(* CoDeSys 2.3.9.48 project: cy-wg-138-006.pro *)
(* Author: Avvitatrice doppia testa *)
(* Libraries: Standard.lib 20.5.14 07:13:26, Iecsfc.lib 16.5.13 13:00:50, SYSLIBCALLBACK.LIB 16.5.13 13:00:50, MBus_03.lib 9.2.13 16:51:58, mod_com.lib 16.5.13 13:00:50, Modb_l05.lib 13.5.15 09:30:08, SerComm.lib 16.5.13 13:00:50, Serial_Interface_01.lib 22.4.13 11:50:14, SysLibEvent.lib 16.5.13 13:00:50, SysLibFile.lib 16.5.13 13:00:50, SysLibPlcCtrl.lib 16.5.13 13:00:50, SysLibRtc.lib 16.5.13 13:00:50, SysLibSockets.lib 22.5.14 15:16:32, Util.lib 16.5.13 13:00:50, WagoLibMBX_01.lib 20.3.12 15:32:40, WagoLibModbus_IP_01.lib 24.7.13 14:05:58 *)

(* PLC configuration (modules and I/O channels)
0750-1506 8DI / 8DO 24V DC 0.5A [Type_34_8_Channels] node 1, in %IB144 out %QB144
  VPN_ST2 AT %IX72.0 [BOOLOnX_I] Ch_1 Digital input
  LAMP_AL AT %QX72.0 [BOOLOnX_Q] Ch_1 Digital output
  KEY_QE_ST AT %IX72.1 [BOOLOnX_I] Ch_2 Digital input
  AT %QX72.1 [BOOLOnX_Q] Ch_2 Digital output
  AT %IX72.2 [BOOLOnX_I] Ch_3 Digital input
  AT %QX72.2 [BOOLOnX_Q] Ch_3 Digital output
  AT %IX72.3 [BOOLOnX_I] Ch_4 Digital input
  AT %QX72.3 [BOOLOnX_Q] Ch_4 Digital output
  AT %IX72.4 [BOOLOnX_I] Ch_5 Digital input
  AT %QX72.4 [BOOLOnX_Q] Ch_5 Digital output
  AT %IX72.5 [BOOLOnX_I] Ch_6 Digital input
  AT %QX72.5 [BOOLOnX_Q] Ch_6 Digital output
  AT %IX72.6 [BOOLOnX_I] Ch_7 Digital input
  AT %QX72.6 [BOOLOnX_Q] Ch_7 Digital output
  AT %IX72.7 [BOOLOnX_I] Ch_8 Digital input
  AT %QX72.7 [BOOLOnX_Q] Ch_8 Digital output
0750-0652#48 RS-232/RS-485 Interface adjustable (48 Bytes) [Type_33_1_Channels] node 2, in %IB96 out %QB96
  AT %IB0 [BYTEOnB_I] First Byte of 48
  AT %QB0 [BYTEOnB_Q] First Byte of 48
0750-0652#48 RS-232/RS-485 Interface adjustable (48 Bytes) [Type_33_1_Channels] node 3, in %IB96 out %QB96
  AT %IB48 [BYTEOnB_I] First Byte of 48
  AT %QB48 [BYTEOnB_Q] First Byte of 48
0750-0652#48 RS-232/RS-485 Interface adjustable (48 Bytes) [Type_33_1_Channels] node 4, in %IB144 out %QB144
  AT %IB96 [BYTEOnB_I] First Byte of 48
  AT %QB96 [BYTEOnB_Q] First Byte of 48
Modbus variables [PFC200MODBUS] node 1, in %IB0 out %QB0 {PlcStopBehaviour = 1; FiledbusErrorBehaviour = 1; TcpOperation = 1; TcpPort = 502; TcpTimeout = 600; UdpOperation = 1; UdpPort = 502; RtuOperation = 0; NodeId = 1; ResponseTimeout = 5000; Interface = 0; Baud = 115200; StopBits = 1; Parity = 1; FlowCtrl = 0; PhysInterface = 0}
Modbus-Master [MB_MASTER] node 2, in %IB0 out %QB0
*)

(* Global variable list: Global_Constants *)
VAR_GLOBAL CONSTANT

	Plant_NAME			: STRING :='cySN:138 cyVER:138 - COIN Genova ';
	Plant_SN			: DWORD  :=138;	(* S/N Impianto di telecontrollo *)
	Plant_SW_VER		: WORD   :=1;		(* Versione SW installata *)


	(* Colour defines *)
	COLOR_RED			: DWORD	:= 16#2020F0;
	COLOR_YELLOW		: DWORD	:= 16#20F0F0;
	COLOR_GREEN			: DWORD	:= 16#20F020;
	COLOR_LIGHT_GREEN	: DWORD := 16#006000;

	(* Parameters *)
	Plant_DefaultTAmb	: INT	:=100;		(* [.1°C] Temperatura ambiente di default in caso di rottura sonda *)
	Plant_MaxRunTAmb	: INT   :=210; 		(* [.1°C] Temperatura ambiente massima funzionamento impianto *)
(*	Plant_AntiFreezeTAmb: INT   :=-40;		(* [.1°C] Antifreeze temperature, start circulators *)
	Plant_VRD_TAlarm	: INT   :=850; 		(* [.1°C] Temperatura di allarme VRD, blocco *)
	Plant_VRD_TMax		: INT   :=800; 		(* [.1°C] Setpoint massimo per uscita VRD *)
	Plant_VRD_TDefault	: INT	:=300;		(* [.1°C] Temperatura di default in caso di errore climatica *)
	Plant_CirOffDelay	: TIME	:=T#30m;	(* (Def.T#15m) Ritardo spegnimento pompe per ricircolo caldaia *)
	Plant_CirOnDelay	: TIME	:=T#15m;
	Plant_MaxWaterLoss	: WORD  :=2;		(* [lt/h] Massima perdita del circuito *) *)

	(* Filesystem *)
	FilesPath  			: STRING :='/media/sd/';(*'S:\'; *)

	(* TCP Logger *)
	Logger_SERVER		: STRING:='';
	Logger_IP			: STRING:='192.168.100.3';
	Logger_PORT			: WORD  :=80;
	Logger_GETSTART		: STRING:='GET /cygmsrv/hsgm.ashx?';
	Logger_GETEND		: STRING:='$R$N$R$N';
	Logger_CHECK		: STRING:='True';
	Logger_CRLF			: STRING:='$R$N';
	Logger_DataFile		: STRING:='/media/sd/LOG.DAT';
	Logger_DataFileOld	: STRING:='/media/sd/LOG.BCK';
	Logger_IndexFile	: STRING:='/media/sd/LOG.IDX';
	Logger_ConnRetries	: BYTE:=5;
	Logger_RecoverMsgs	: BYTE:=25;

	(* TCP Remote *)
	Remote_PORT			: WORD  :=10;
	Remote_WELCOME		: STRING:='Connected$R$N';
	Remote_OK			: STRING:='OK$R$N';
	Remote_ERROR		: STRING:='ERROR$R$N';

	(* TCP Sockets *)
	MAX_SEND_TCP_SERVER					 : DWORD:=60000;(*60000*)
	MAX_RECEIVE_TCP_SERVER				 : DWORD:=10000;
	MAX_RECEIVE_TCP_SERVER_SOCKET	 	 : DWORD:=2500;
	MAX_SEND_TCP_CLIENT					 : DWORD:=30000;(*15000*)
	MAX_RECEIVE_TCP_CLIENT				 : DWORD:=2500;
	MAX_RECEIVE_TCP_CLIENT_SOCKET		 : DWORD:=2500;
	MAX_RECEIVE_UDP_SERVER				 : INT  :=1472;
	MAX_RECEIVE_UDP_CLIENT				 : INT  :=1472;
	CONNECT_WATCHDOG_TIME				 : TIME :=t#10s;

END_VAR


VAR_GLOBAL
(*	TestNodoInterogato: BYTE;
	NodoDaInterrogare: BYTE;
	InibiscoModbus: BOOL;
 *)

	NodoDaInterrogareChiller: BYTE;
	InibiscoModbusChiller: BOOL;
	NodoDaInterrogareANZ: BYTE;
	InibiscoModbusANZ: BOOL;

	NodoDaInterrogareMB2: BYTE;
	InibiscoModbusMB2: BOOL;

	NodoDaInterrogareMB1: BYTE;
	InibiscoModbusMB1: BOOL;

	NodoDaInterrogareMB3: BYTE;
	InibiscoModbusMB3: BOOL;


END_VAR

VAR_GLOBAL RETAIN
	cmd_ControlMode_UTA01: BOOL;		(* variabili per abilitazione controllo UTA da CRONO o con comandi manuali da registro Modbus *)
	cmd_ControlMode_UTA02: BOOL;		(* variabili per abilitazione controllo UTA da CRONO o con comandi manuali da registro Modbus *)
	cmd_ControlMode_UTA03: BOOL;		(* variabili per abilitazione controllo UTA da CRONO o con comandi manuali da registro Modbus *)
	cmd_ControlMode_UTA04: BOOL;		(* variabili per abilitazione controllo UTA da CRONO o con comandi manuali da registro Modbus *)
	cmd_ControlMode_UTA05: BOOL;		(* variabili per abilitazione controllo UTA da CRONO o con comandi manuali da registro Modbus *)
	cmd_ControlMode_UTA06: BOOL;		(* variabili per abilitazione controllo UTA da CRONO o con comandi manuali da registro Modbus *)
	cmd_ControlMode_UTA07: BOOL;		(* variabili per abilitazione controllo UTA da CRONO o con comandi manuali da registro Modbus *)
	cmd_ControlMode_UTA08: BOOL;		(* variabili per abilitazione controllo UTA da CRONO o con comandi manuali da registro Modbus *)
	cmd_ControlMode_UTA09: BOOL;		(* variabili per abilitazione controllo UTA da CRONO o con comandi manuali da registro Modbus *)
	cmd_ControlMode_UTA10: BOOL;		(* variabili per abilitazione controllo UTA da CRONO o con comandi manuali da registro Modbus *)
	cmd_ControlMode_UTA12: BOOL;		(* variabili per abilitazione controllo UTA da CRONO o con comandi manuali da registro Modbus *)
	cmd_ControlMode_UTA13: BOOL;		(* variabili per abilitazione controllo UTA da CRONO o con comandi manuali da registro Modbus *)

END_VAR

(* Global variable list: Global_Retain *)
VAR_GLOBAL RETAIN PERSISTENT
(*	Mode_Manual : BOOL := FALSE; *)


(*	VRD01_Clima : typ_Clima;
	VRD02_Clima : typ_Clima;
	VRD03_Clima : typ_Clima;
	VRD04_Clima : typ_Clima; *)

	CHI01_Clima	: typ_Clima;
	CHI02_Clima	: typ_Clima;


(*	Ctl01_Counter	:	DWORD;
	Ctl02_Counter	:	DWORD; *)

(* Impostazioni di imipanto *)
(*
	DelayAllarmeTemperaturaNonRaggiunta: INT:=60;
	DeltaInterventoAllarmeTempeaturaNonRaggiuta: INT:=400;
	OffsetSetPointManuale:INT:=50;							(* Offset al Setpoint manuale per comensare lo scambiatore *)

	SogliaMinStartAntigelo: INT:=50;
	SogliaMinStopAntigelo: INT:=80;
	BitAbilitaAntigelo: BOOL:=TRUE;
*)

END_VAR

(* Global variable list: Global_Variables *)
VAR_GLOBAL

	SYS    : typ_SYS;
	Logger : typ_Logger;

	Lamp	:	LAMP_AL_GENERALE; (* Per gestione allarme generico impianto *)

	(**** PLANT OBJECTS ****)

	(* Frigo *)
	CHIAERMEC01	:obj_MODBUS_FRG_AER485P1 := (ID:=1, Address:=1);
	CHIAERMEC02	:obj_MODBUS_FRG_AER485P1 := (ID:=2, Address:=2);

	(* Cronothermostat *)
	THER01	:	obj_CRONTER_01 := (ID:=1, Local_MaxRunTAmb:=250,Histeresys:=10);
	THER02	:	obj_CRONTER_01 := (ID:=2, Local_MaxRunTAmb:=250,Histeresys:=10);
	THER03	:	obj_CRONTER_01 := (ID:=3, Local_MaxRunTAmb:=250,Histeresys:=10);
	THER04	:	obj_CRONTER_01 := (ID:=4, Local_MaxRunTAmb:=250,Histeresys:=10);
	THER05	:	obj_CRONTER_01 := (ID:=5, Local_MaxRunTAmb:=250,Histeresys:=10);
	THER06	:	obj_CRONTER_01 := (ID:=6, Local_MaxRunTAmb:=250,Histeresys:=10);
	THER07	:	obj_CRONTER_01 := (ID:=7, Local_MaxRunTAmb:=250,Histeresys:=10);
	THER08	:	obj_CRONTER_01 := (ID:=8, Local_MaxRunTAmb:=250,Histeresys:=10);
	THER09	:	obj_CRONTER_01 := (ID:=9, Local_MaxRunTAmb:=250,Histeresys:=10);
	THER10	:	obj_CRONTER_01 := (ID:=10, Local_MaxRunTAmb:=250,Histeresys:=10);
	THER12	:	obj_CRONTER_01 := (ID:=12, Local_MaxRunTAmb:=250,Histeresys:=10);
	THER13	:	obj_CRONTER_01 := (ID:=13, Local_MaxRunTAmb:=250,Histeresys:=10);


	CronEd	: 	obj_CRON_EDITOR_01;

	(* Gateway sonde Zeegbe *)

	GATEWAY	:	obj_GATEWAY_01 := (ID:=1, address:=1); 	(* gate way  *)


(* Sonde Tmperatura *)

	ZTHL01	:	obj_ZTHL_01 := (ID:=1, address:=16); 	(* Piano sotterraneo Rep. Bambino  *)
	ZTHL02	:	obj_ZTHL_01 := (ID:=2, address:=17); 	(* Piano sotterraneo Rep. Donna  *)
	ZTHL03	:	obj_ZTHL_01 := (ID:=3, address:=18); 	(* Piano terra ingresso - profumi   *)
	ZTHL04	:	obj_ZTHL_01 := (ID:=4, address:=19); 	(* Piano terra ingresso - rep. Uomo    *)
	ZTHL05	:	obj_ZTHL_01 := (ID:=5, address:=20);	(* Piano primo - reparto casa - lato cucina *)
	ZTHL06	:	obj_ZTHL_01 := (ID:=6, address:=21);	(* Piano primo - reparto casa - lato casse - uffici *)

(* Sonde CO2 *)

	COOV01	:	obj_COOV_01 := (ID:=1, address:=31); 	(* Piano sotterraneo Rep. Bambino  *)
	COOV02	:	obj_COOV_01 := (ID:=2, address:=32);	(* Piano sotterraneo Rep. Donna  *)
	COOV03	:	obj_COOV_01 := (ID:=3, address:=33);	(* Piano terra ingresso - profumi   *)
	COOV04	:	obj_COOV_01 := (ID:=4, address:=34);	(* Piano terra ingresso - rep. Uomo    *)
	COOV05	:	obj_COOV_01 := (ID:=5, address:=35);	(* Piano primo - reparto casa - lato cucina *)
	COOV06	:	obj_COOV_01 := (ID:=6, address:=36);	(* Piano primo - reparto casa - lato casse - uffici *)


	ANZ01	:	obj_MODBUS_FRER_QUBOH:= (ID:=1,Address:=1);	(* Generale  *)
	ANZ02	:	obj_MODBUS_FRER_QUBOH := (ID:=2,Address:=2);	(* QE. Uffici - QU  *)
	ANZ03	:	obj_MODBUS_FRER_QUBOH:= (ID:=3,Address:=3);	(* Gruppo frigo 1  *)
	ANZ04	:	obj_MODBUS_FRER_QUBOH:= (ID:=4,Address:=4);	(* Gruppo frigo 2  *)
	ANZ05	:	obj_MODBUS_FRER_QUBOH:= (ID:=5,Address:=5);	(* Q.E. UTA 1-5  *)
	ANZ06	:	obj_MODBUS_FRER_QUBOH:= (ID:=6,Address:=6);	(* Linee UTA (n.3 - una per fase) *)
	ANZ07	:	obj_MODBUS_FRER_QUBOH:= (ID:=7,Address:=7);	(* Linee UTA (n.3 - una per fase) *)
	ANZ08	:	obj_MODBUS_FRER_QUBOH:= (ID:=8,Address:=8);	(* Linee UTA (n.2 - una per fase) *)


	TREND : obj_MODBUS_TRENDCOIN_01 := (ID:=1,Address:=1);


(*** UTA ***)

	UTA01  	: obj_UTA_02:=(ID:=1);
	UTA02  	: obj_UTA_02:=(ID:=2);
	UTA03  	: obj_UTA_02:=(ID:=3);
	UTA04  	: obj_UTA_02:=(ID:=4);
	UTA05  	: obj_UTA_02:=(ID:=5);
	UTA06  	: obj_UTA_02:=(ID:=6);
	UTA07  	: obj_UTA_02:=(ID:=7);
	UTA08  	: obj_UTA_02:=(ID:=8);
	UTA09  	: obj_UTA_02:=(ID:=9);
	UTA10  	: obj_UTA_02:=(ID:=10);
(*	UTA11  	: obj_UTA_02:=(ID:=11); *)
	UTA12  	: obj_UTA_02:=(ID:=12);
	UTA13  	: obj_UTA_02:=(ID:=13);


	(** Communication **)
	(* ModBus *)

	MODB01	:	obj_MODBUS		:= (ID:=1, COM:=0, BAUDRATE:=BAUD_19200,RS485:=TRUE,MB_timeOut:=t#500ms);
	MODB02	:	obj_MODBUS		:= (ID:=2, COM:=2, BAUDRATE:=BAUD_9600 ,N_STOPBits:=2,RS485:=TRUE,MB_timeOut:=t#500ms);
	MODB03	:	obj_MODBUS 		:= (ID:=3, COM:=3, BAUDRATE:=BAUD_19200,N_STOPBits:=2,RS485:=TRUE,MB_timeOut:=t#500ms);
	MODB04	:	obj_MODBUS 		:= (ID:=4, COM:=4, BAUDRATE:=BAUD_19200,N_STOPBits:=2,RS485:=TRUE,MB_timeOut:=t#500ms);


	(**** SIMULATION ONLY ****)

	AggiornaLog: BOOL;

	(*...*)


END_VAR

(* Data type in Logger *)
TYPE en_Logger_ErrLev :
(
	EL_Log			:=0,
	EL_Wrn			:=1,
	EL_Alarm		:=2,
	EL_AlarmStop	:=3
);
END_TYPE

(* Data type in Logger *)
TYPE en_Logger_Status :
(
	S_Logger_UNKNOWN := 0,
	S_Logger_IDLE,
	S_Logger_WAITCONN,
	S_Logger_WAITTX,
	S_Logger_WAITRESP,
	S_Logger_ERROR
);
END_TYPE

(* Data type *)
TYPE en_SYS_Objects :
(
	EO_SYS		:=0,  (* PLC *)
	EO_VPN		:=1,  (* VPN *)
	EO_DOOR		:=2,  (* Door & access control *)

	EO_CAL		:=10, (* Caldaia *)
	EO_CIR		:=11, (* Circolatore *)
	EO_CRON		:=12, (* Crono-termostato *)
	EO_VRD		:=13, (* Valvola miscelatore pannelli *)
	EO_CTL		:=14, (* Contalitri *)
	EO_CTB		:=15, (* Contabilizzatore *)
	EO_TPV		:=16, (* Temperature probes values *)
	EO_PPV		:=17, (* Pressure probes values *)
	EO_PBV		:=18, (* Over-Pressure Alarms *)
	EO_TBV		:=19, (* Over-Temperature Alarms *)
	EO_PMV		:=20, (* Under-Pressure Alarms *)
	EO_GRU		:=21, (* Gruppo termico *)
	EO_PDC		:=22, (* Pompa di calore *)
	EO_SOL		:=23, (* Pannello solare termico *)
	EO_ESOL		:=24, (* Pannello solare fotovoltaico *)
	EO_GAS		:=25, (* Contatore GAS *)
	EO_PORT		:=26, (* Misuratore di portata *)
	EO_FPV		:=27, (* Flow probes values *)
	EO_ANZ		:=28, (* Analizzatore di rete *)
	EO_SCA		:=29, (* Signal Control Alarms *)
	EO_LUX		:=30, (* Base Illumination point *)
	EO_LUXM		:=31, (* Metered Illumination point *)
	EO_PSG		:=32, (* Sensore di passaggio *)
	EO_HVAC		:=33, (* Heating, Ventilating and Air Conditioning *)
	EO_HYGRV	:=34, (* Relative Humidity sensors value *)
	EO_COOV		:=35, (* Carbon Dioxide CO2 sensors value *)
	EO_INV		:=36, (* Inverter *)
	EO_STR		:=37, (* Smart string box *)

	EO_CIRD		:=39, (* Double CIR *)
	EO_ACS		:=40, (* Hot domestic water *)
	EO_CHI		:=41, (* Chiller *)
	EO_THER		:=42, (* Thermostat *)
	EO_CIRM		:=43, (* Modbus CIR *)
	EO_CIRDM	:=44, (* Modbus double CIR *)


	EO_UTA		:=47, (* UTA  *)
	EO_CHIAERMEC:=48, (* Frigorifero Aermec *)
	EO_UTACOIN	:=49, (* UTA  *)
	EO_POOL	:=50, 		(* Mischiotto  *)
	EO_ZCOOV:= 51, 		(*Sonda C02 Zigbee ZCOOVxxx *)


	EO_ZGW			:=200,  (* ZigBee - Gateway *)
	EO_ZRM			:=201,	(* ZigBee - Repeater *)
	EO_ZREL			:=202,	(* ZigBee - Actuator rele *)
	EO_ZTHL			:=203,	(* ZigBee - Temperature Sensor *)

	EO_ASGW			:=250,	(* ASi - Gateway *)
	EO_ASCBI		:=251,	(* ASi - Input Board, Ciabatta *)

	EO_LON			:=1000, (* Bus - LON *)
	EO_MODBUS		:=1001, (* Bus - MODBUS *)
	EO_MBUS			:=1002, (* Bus - M-BUS *)
	EO_MODBUS_TCP	:=1003, (* Bus - MODBUS TCP *)

	EO_GENERIC		:=9000, (* Generic dataset *)
	EO_EXPO			:=9001 (* EXPO dataset *)
);
END_TYPE

(* Data type *)
TYPE en_SYS_Status :
(
	S_UNKNOWN  := 0,
	S_STARTUP,
	S_INIT_RTC,
	S_INIT_VAR,
	S_AUTOTEST,
	S_RUNNING,
	S_SHUTDOWN,
	S_HALT
);
END_TYPE

(* Data type in Plant_Objects *)
TYPE typ_Clima : (* CURVA CLIMATICA *)
STRUCT
	InitOK:		BOOL;
	Points: 	ARRAY [0..10] OF POINT;
END_STRUCT
END_TYPE

(* Data type in Plant_Objects *)
TYPE typ_Cron_Calendar :
STRUCT
	Profile		: ARRAY[0..384] OF BYTE;
END_STRUCT
END_TYPE

(* Data type in Plant_Objects *)
TYPE typ_Cron_Jolly :
STRUCT
	Start		: DT;
	End			: DT;
	Temp		: WORD;
	Flags		: WORD; (* B0:Enabled B1..B15:Unused *)
END_STRUCT
END_TYPE

(* Data type in Plant_Objects *)
TYPE typ_Cron_Profile :
STRUCT
	Flags		: WORD;
	Setpoint	: ARRAY [0..95] OF WORD;
END_STRUCT
END_TYPE

(* Data type in Plant_Objects *)
TYPE typ_Frigo :
STRUCT
	Status	:	BOOL;		(* 0=OFF, 1=ON	*)
	Mode	:	BOOL;		(* 0=COLD, 1=HOT	*)
	Reset	:	BOOL;		(* 1=RESET	*)

	Alarm	:	DWORD;		(* 30 alarms of type bool grouped in one variable of 32 bits (last 2 don't used) *)

	(*  ALARM CODE (bit order of dword "Alarm": first is bit 0, last bit29)
        8	:	Allarme flussostato
		9	:	Allarme termica pompa condensante 
		10	:	Allarme termica pompa evaporante 
		11	:	Allarme resa 
		12	:	Allarme termica compressore circuito 1 
		13	:	Allarme bassa pressione circuito 1
		14	:	Allarme alta pressione circuito 1 
		15	:	Allarme antigelo circuito 1	
		16	:	Allarme termica ventilatore circuito 1	
		17	:	Allarme pressostato olio crcuito 1	
		18	:	Allarme sonda circuito 1	
		19	:	Allarme termica compressore circuito 2	
		20	:	Allarme bassa pressione circuito 2	
		21	:	Allarme alta pressione circuito 2	
		22	:	Allarme antigelo circuito 2	
		23	:	Allarme termica ventilatore circuito 2	
		24	:	Allarme pressostato olio circuito 2	
		25	:	Allarme sonda circuito 2	
		26	:	Allarme monitor tensione	
		27	:	Allarme pumpdown circuito 1	
		28	:	Allarme pumpdown circuito 2	
		29	:	Allarme eeprom	
		30	:	Allarme clock calendar	
		80	:	Allarme flussostato recuperatore	
		81	:	Allarme termica compressore circuito 1A	
		82	:	Allarme termica compressore circuito 1B	
		83	:	Allarme termica pompa evaporatore 1	
		84	:	Allarme termica pompa evaporatore 2	
		85	:	Allarme termica pompa evaporatore 3	
		86	:	Allarme antigelo evaporatore circuito 1	
		87	:	Allarme antigelo evaporatore circuito 2	
	*)


END_STRUCT
END_TYPE

(* Data type in Logger *)
TYPE typ_Logger :
STRUCT
	Status		: en_Logger_Status;

	SendReq		: BOOL;
	SendIdx		: DWORD;
	SendData	: ARRAY [0..MAX_SEND_TCP_CLIENT] OF BYTE;
	SendLen		: DINT;

	TData		: ARRAY [0..MAX_SEND_TCP_CLIENT] OF BYTE;
	TLen		: DINT;

	LastIdxPos	: DWORD;

	(* Temporary variables used by objects *)
	s1			: STRING(256);
	i1			: WORD;

END_STRUCT
END_TYPE

(* Data type in Plant_Objects *)
TYPE typ_MODBUS_CIR :
STRUCT
	PumpStatus		:	WORD;
	PumpFault		:	BOOL;
	PumpBoardTemp	:	INT;	(* Electonic board temperature  [°C] *)
	PumpVoltage		:	WORD;	(* Input voltage rms [V] *)
	PumpCurrent		:	WORD;	(* Output current [E-3 A]	*)
	PumpRPM			:	WORD;	(* Round per minute [rpm] *)
	PumpPower		:	WORD;	(* Power [W] *)
	PumpOpTime		:	DWORD;	(* Pump operating time [h] *)
	PumpHead		:	WORD;	(* [E-1 m] *)
	PumpFlow		:	WORD;	(* Extimated flow [E-1 m3/h] *)
	PumpLiqTemp		:	WORD;	(* Liquid temperature [°C] *)
	PumpAlarm		:	ARRAY [0..14] OF WORD;

END_STRUCT
END_TYPE

(* Data type in Plant_Objects *)
TYPE typ_MODBUS_FRER_QUBOH :
STRUCT
	V_L1N		:	DINT;	(* E-3 V *)
	V_L2N		:	DINT;
	V_L3N		:	DINT;
	V_L1L2		:	DINT;
	V_L2L3		:	DINT;
	V_L3L1		:	DINT;
	I_L1			:	DINT;	(* E-3 A *)
	I_L2			:	DINT;
	I_L3			:	DINT;

	FREQ		:	DWORD;	(* E-3 Hz *)

	P_3P			:	DINT;	(* W *)
	Q_3P		:	DINT;	(* VAr *)
	PF_3P		:	DINT;	(* E-3 *)
	WH_3P		:	DINT;	(* Wh *)
	VARH_3P		:	DINT;	(* VArh *)
	Multiplier	:	DWORD;

	V_3P		:	DINT;	(* E-3 V *)
	I_3P		:	DINT;	(* E-3 A *)

	COS_3P		:	DINT;	(* E-3 *)

	VA_3P		:	DINT;	(* VA *)
	P_L1		:	DWORD;	(* W *)
	P_L2		:	DWORD;
	P_L3		:	DWORD;
	Q_L1		:	DINT;	(* VAr *)
	Q_L2		:	DINT;
	Q_L3		:	DINT;
	VA_L1		:	DINT;	(* VA *)
	VA_L2		:	DINT;
	VA_L3		:	DINT;
	PF_L1		:	DINT;	(* E-3 *)
	PF_L2		:	DINT;
	PF_L3		:	DINT;
	COS_L1		:	DINT;	(* E-3 *)
	COS_L2		:	DINT;
	COS_L3		:	DINT;

	P_3P_Max	:	DINT;	(* W *)
	P_3P_Avg		:	DINT;

	I_L1_Max	:	DINT;	(* E-3 A *)
	I_L2_Max	:	DINT;
	I_L3_Max	:	DINT;

	Q_3P_Max	:	DINT;	(* VAr *)

END_STRUCT
END_TYPE

(* Data type in Plant_Objects *)
TYPE typ_MODBUS_VAR : (* Gestione parametri MODBUS *)
STRUCT
	SlaveAddress	: BYTE;
	FunCode			: BYTE;
	FunAddress		: WORD;
	Refresh_Time	: BYTE; (* 0:No refresh x:Refresh in seconds *)
	Refresh_Cnt		: BYTE; (* INTERNAL *)
	Variable		: POINTER TO WORD;
	Variable_Size	: BYTE;
	Variable_Mirror : WORD; (* INTERNAL [Force refresh on read variables when <>0] *)
END_STRUCT
END_TYPE

(* Data type *)
TYPE typ_SYS :
STRUCT
	Status			: en_SYS_Status;
	Warning			: BOOL;
	Alarm			: BOOL;
	AlarmStop		: BOOL;

	Time_LogString	: STRING;
	Time_Year		: WORD;
	Time_Month		: BYTE;
	Time_Day		: BYTE;
	Time_Hour		: BYTE;
	Time_Minute		: BYTE;

	Time_CT_DT		: DT;
	Time_CT_Day		: WORD;
	Time_CT_Quarter	: BYTE;

	LastLogs_Idx	: BYTE;
	LastLogs_Dat	: ARRAY[0..5] OF STRING;
	LastLogs_Msg	: ARRAY[0..5] OF STRING;

END_STRUCT
END_TYPE

(* Data type in Plant_Objects *)
TYPE typ_VisuStrutturaMbus :
STRUCT

	sdNodoPresente: STRING(16);
	sdEnergia: STRING(16);
	sdPotenza: STRING(16);
	sdVolume: STRING(16);
	sdFlow: STRING(16);
	sdTempIngresso: STRING(8);
	sdTempaUscita: STRING(8);
	sdTempDelta: STRING(8);

END_STRUCT
END_TYPE

(* POU PLC_PRG, ST *)
PROGRAM PLC_PRG
VAR
	Timer1: TON; (* Fast controls tick *)
	Timer2: TON; (* Plant control tick *)
	Timer3: TON; (* Logger timer *)

	i : INT;

	R_TRIG_CHIAERMEC01_ScriviDato: F_TRIG;
	R_TRIG_CHIAERMEC02_ScriviDato: F_TRIG;
	R_TRIG_TREND_ScriviDato: F_TRIG;

	aggiornalogdaModBus: BOOL;
	tonaggiornaLogdaModBus: TON;
	EseguiLog: INT;
	Ton_pausaTrig: TON;
	s1: STRING;
	R_TrigAggiornaLog: R_TRIG;
	allarme,warning:BOOL;
END_VAR
VAR_INPUT
	RichiestaLogDaRemoto: BOOL;
END_VAR
(******************************************************************************
 ****                           MAIN TASK CODE                             ****
 ******************************************************************************

	Network setup:
		IP  = 192.168.100.2 | MSK = 255.255.255.0
		GW	= 192.168.100.1 | DNS = 192.168.100.1
		SNTP = 193.204.114.232 (3600s) ==> 192.168.100.3

*)

(*==============================*)
(*===== Main status machine ====*)
(*==============================*)
Main_Stm();

(*==============================*)
(*== Running cycle operations ==*)
(*==============================*)
IF SYS.Status>S_INIT_VAR THEN
	(* Execute cycle processes *)


	MODB01();
(*	TREND(ModBus:=MODB01,
			ScriviRUN_UTA01:=UTA01.cmd_DO_OUT,
			ScriviRUN_UTA02:=UTA02.cmd_DO_OUT,
			ScriviRUN_UTA03:=UTA03.cmd_DO_OUT,
			ScriviRUN_UTA04:=UTA04.cmd_DO_OUT,
			ScriviRUN_UTA05:=UTA05.cmd_DO_OUT,
			ScriviRUN_UTA06:=UTA06.cmd_DO_OUT,
			ScriviRUN_UTA07:=UTA07.cmd_DO_OUT,
			ScriviRUN_UTA08:=UTA08.cmd_DO_OUT,
			ScriviRUN_UTA09:=UTA09.cmd_DO_OUT,
			ScriviRUN_UTA10:=UTA10.cmd_DO_OUT,
			ScriviRUN_UTA12:=UTA12.cmd_DO_OUT,
			ScriviRUN_UTA13:=UTA13.cmd_DO_OUT,
			); *)




	TREND(ModBus:=MODB01);

	TREND(
			ControlMode_UTA01:=cmd_ControlMode_UTA01,
 			ControlMode_UTA02:=cmd_ControlMode_UTA02,
			ControlMode_UTA03:=cmd_ControlMode_UTA03,
			ControlMode_UTA04:=cmd_ControlMode_UTA04,
			ControlMode_UTA05:=cmd_ControlMode_UTA05,
			ControlMode_UTA06:=cmd_ControlMode_UTA06,
			ControlMode_UTA07:=cmd_ControlMode_UTA07,
			ControlMode_UTA08:=cmd_ControlMode_UTA08,
			ControlMode_UTA09:=cmd_ControlMode_UTA09,
			ControlMode_UTA10:=cmd_ControlMode_UTA10,
			ControlMode_UTA12:=cmd_ControlMode_UTA12,
			ControlMode_UTA13:=cmd_ControlMode_UTA13,
			ScriviRUN_UTA01:=UTA01.cmd_DO_OUT ,
			ScriviRUN_UTA02:=UTA02.cmd_DO_OUT ,
			ScriviRUN_UTA03:=UTA03.cmd_DO_OUT ,
			ScriviRUN_UTA04:=UTA04.cmd_DO_OUT ,
			ScriviRUN_UTA05:=UTA05.cmd_DO_OUT ,
			ScriviRUN_UTA06:=UTA06.cmd_DO_OUT ,
			ScriviRUN_UTA07:=UTA07.cmd_DO_OUT ,
			ScriviRUN_UTA08:=UTA08.cmd_DO_OUT ,
			ScriviRUN_UTA09:=UTA09.cmd_DO_OUT ,
			ScriviRUN_UTA10:=UTA10.cmd_DO_OUT ,
			ScriviRUN_UTA12:=UTA12.cmd_DO_OUT ,
			ScriviRUN_UTA13:=UTA13.cmd_DO_OUT ,
			ScriviSP_UTA01:=UTA01.cmd_DO_SetPoint ,
			ScriviSP_UTA02:=UTA02.cmd_DO_SetPoint ,
			ScriviSP_UTA03:=UTA03.cmd_DO_SetPoint ,
			ScriviSP_UTA04:=UTA04.cmd_DO_SetPoint ,
			ScriviSP_UTA05:=UTA05.cmd_DO_SetPoint ,
			ScriviSP_UTA06:=UTA06.cmd_DO_SetPoint ,
			ScriviSP_UTA07:=UTA07.cmd_DO_SetPoint ,
			ScriviSP_UTA08:=UTA08.cmd_DO_SetPoint ,
			ScriviSP_UTA09:=UTA09.cmd_DO_SetPoint ,
			ScriviSP_UTA10:=UTA10.cmd_DO_SetPoint ,
			ScriviSP_UTA12:=UTA12.cmd_DO_SetPoint ,
			ScriviSP_UTA13:=UTA13.cmd_DO_SetPoint ,
			ModBus:=MODB01 ,
			Status_Log=> ,
			Status_Vis=> );


	NodoDaInterrogareMB1:=1;

UTA01(
	UTA_ST:=TREND.MB_BitStatoCoil[19],
	UTA_CentrAL:=TREND.MB_BitStato[102] OR TREND.MB_BitStato[103],   (* TRUE= Flusso , FALSE = No Flusso *)
	T_AMB:=TREND.MB_RegistriLetti[134] ,
	UR_AMB:=TREND.MB_RegistriLetti[135]  ,
	T_MISC:=TREND.MB_RegistriLetti[136]  ,
	UR_MISC:=TREND.MB_RegistriLetti[137]  ,
	T_MAND:=TREND.MB_RegistriLetti[138]  ,
	T_EST:=TREND.MB_RegistriLetti[139]  ,
	UR_EST:= TREND.MB_RegistriLetti[140] ,
	ENTALPIA_EST:=TREND.MB_RegistriLetti[141]  ,
	ENTALPIA_AMB:=TREND.MB_RegistriLetti[142] ,
	UMID_ASS_EST:=TREND.MB_RegistriLetti[143]  ,
	UMID_ASS_AMB:= TREND.MB_RegistriLetti[144] ,
	UMID_ASS_MISC:=TREND.MB_RegistriLetti[145] ,
	UMID_ASS_CONDEN:=TREND.MB_RegistriLetti[146]  ,
	SET_COMP_T_AMB:=TREND.MB_RegistriLetti[147]  ,
	RITAR_SET_T_AMB:= TREND.MB_RegistriHoldingLetti[68],
	SET_T_MAND:= TREND.MB_RegistriHoldingLetti[69] ,
	SET_ANTIGELO:= TREND.MB_RegistriHoldingLetti[70] ,
	SET_UR_AMB:= TREND.MB_RegistriHoldingLetti[71],
	ISTERESI_UR_AMB:= TREND.MB_RegistriHoldingLetti[72] ,
	SET_F_ANTIG_AMB:= TREND.MB_RegistriHoldingLetti[73] ,
	SOGLIA_T_EST_VR:=  TREND.MB_RegistriHoldingLetti[74],
	MIN_AP_SERR_E_R:=  TREND.MB_RegistriHoldingLetti[75],
	MIN_AP_SERR_ESP:=  TREND.MB_RegistriHoldingLetti[76],
	RID_SET_T_RISC:=  TREND.MB_RegistriHoldingLetti[77],
	VENT_MAND:= TREND.MB_BitStato[141],
	VENT_RIPR:=TREND.MB_BitStato[142] ,
	P_UMIDIF:=TREND.MB_BitStato[143] ,
	VALV_B_FREDDA:=TREND.MB_BitStato[151] ,
	VALV_B_CALDA:=TREND.MB_BitStato[152] ,
	SERRANDE_ESP:= TREND.MB_BitStato[153],
	SERRAND_EST_RIC:= TREND.MB_BitStato[154],
	ABILITA:=TREND.MB_BitStatoCoil[19] ,
	STATO_VENT_M:=TREND.MB_BitStato[99] ,
	STATO_VENT_R:=TREND.MB_BitStato[100] ,
	FILTRO:=TREND.MB_BitStato[101] ,
	FLUSSO_VM:=TREND.MB_BitStato[102] ,
	FLUSSO_VR:= TREND.MB_BitStato[103],
	FILTRI_INTASATI:= TREND.MB_BitStato[104],
	ALL_VERIFICA_VM:=TREND.MB_BitStato[105] ,
	ALL_VERIFICA_VR:= TREND.MB_BitStato[106],
	ALL_V011_MANC_SPEGN:= TREND.MB_BitStato[107],
	ALL_V011_MANC_FUNZ:=TREND.MB_BitStato[108],
	ALL_V012_MANC_SPEGN:=TREND.MB_BitStato[109] ,
	ALL_V012_MANC_FUNZ:=TREND.MB_BitStato[110],
	cmd_DI_RUN:=THER01.RunCrono,
	cmd_DI_SetPoint:=THER01.SetPoint,
	UTA_CONTROL_MODE:=cmd_ControlMode_UTA01	);



	UTA02(
	UTA_ST:= TREND.MB_BitStatoCoil[20],     	(* ABILITA UTA  *)
	UTA_CentrAL:=TREND.MB_BitStato[120] OR TREND.MB_BitStato[121],	 (* TRUE= Flusso , FALSE = No Flusso *)
	T_AMB:=TREND.MB_RegistriLetti[155] ,
	UR_AMB:=TREND.MB_RegistriLetti[156]  ,
	T_MISC:=TREND.MB_RegistriLetti[157]  ,
	UR_MISC:=TREND.MB_RegistriLetti[158]  ,
	T_MAND:=TREND.MB_RegistriLetti[159]  ,
	T_EST:=TREND.MB_RegistriLetti[165]  ,
	UR_EST:= TREND.MB_RegistriLetti[166] ,
	ENTALPIA_EST:=TREND.MB_RegistriLetti[169]  ,
	ENTALPIA_AMB:=TREND.MB_RegistriLetti[170] ,
	UMID_ASS_EST:=TREND.MB_RegistriLetti[171]  ,
	UMID_ASS_AMB:= TREND.MB_RegistriLetti[172] ,
	UMID_ASS_MISC:=TREND.MB_RegistriLetti[173] ,
	UMID_ASS_CONDEN:=TREND.MB_RegistriLetti[174]  ,
	SET_COMP_T_AMB:=TREND.MB_RegistriLetti[167]  ,
	RITAR_SET_T_AMB:= TREND.MB_RegistriHoldingLetti[78],
	SET_T_MAND:= TREND.MB_RegistriHoldingLetti[79] ,
	SET_ANTIGELO:= TREND.MB_RegistriHoldingLetti[80] ,
	SET_UR_AMB:= TREND.MB_RegistriHoldingLetti[81],
	ISTERESI_UR_AMB:= TREND.MB_RegistriHoldingLetti[82] ,
	SET_F_ANTIG_AMB:= TREND.MB_RegistriHoldingLetti[83] ,
	SOGLIA_T_EST_VR:=  TREND.MB_RegistriHoldingLetti[84],
	MIN_AP_SERR_E_R:=  TREND.MB_RegistriHoldingLetti[85],
	MIN_AP_SERR_ESP:=  TREND.MB_RegistriHoldingLetti[86],
	RID_SET_T_RISC:=  TREND.MB_RegistriHoldingLetti[87],
	VENT_MAND:= TREND.MB_BitStato[111],
	VENT_RIPR:=TREND.MB_BitStato[112] ,
	P_UMIDIF:=TREND.MB_BitStato[113] ,
	VALV_B_FREDDA:=TREND.MB_BitStato[181] ,
	VALV_B_CALDA:=TREND.MB_BitStato[182] ,
	SERRANDE_ESP:= TREND.MB_BitStato[183],
	SERRAND_EST_RIC:= TREND.MB_BitStato[184],
	ABILITA:=TREND.MB_BitStatoCoil[20] ,
	STATO_VENT_M:=TREND.MB_BitStato[117] ,
	STATO_VENT_R:=TREND.MB_BitStato[118] ,
	FILTRO:=TREND.MB_BitStato[119] ,
	FLUSSO_VM:=TREND.MB_BitStato[120] ,
	FLUSSO_VR:= TREND.MB_BitStato[121],
	FILTRI_INTASATI:= TREND.MB_BitStato[127],
	ALL_VERIFICA_VM:=TREND.MB_BitStato[128] ,
	ALL_VERIFICA_VR:= TREND.MB_BitStato[129],
	ALL_V011_MANC_SPEGN:= TREND.MB_BitStato[130],
	ALL_V011_MANC_FUNZ:=TREND.MB_BitStato[131],
	ALL_V012_MANC_SPEGN:=TREND.MB_BitStato[132] ,
	ALL_V012_MANC_FUNZ:=TREND.MB_BitStato[133],
	cmd_DI_RUN:=THER02.RunCrono,
	cmd_DI_SetPoint:=THER02.SetPoint,
	UTA_CONTROL_MODE:=cmd_ControlMode_UTA02	);





	UTA03(
	UTA_ST:= TREND.MB_BitStatoCoil[21],     	(* V021 VENT.MAND.UTA2  *)
	UTA_CentrAL:=TREND.MB_BitStato[125] OR TREND.MB_BitStato[126],	 (* TRUE= Flusso , FALSE = No Flusso *)
	T_AMB:=TREND.MB_RegistriLetti[160] ,
	UR_AMB:=TREND.MB_RegistriLetti[161]  ,
	T_MISC:=TREND.MB_RegistriLetti[162]  ,
	UR_MISC:=TREND.MB_RegistriLetti[163]  ,
	T_MAND:=TREND.MB_RegistriLetti[164]  ,
	T_EST:=TREND.MB_RegistriLetti[165]  ,
	UR_EST:= TREND.MB_RegistriLetti[166] ,
	ENTALPIA_EST:=TREND.MB_RegistriLetti[169]  ,
	ENTALPIA_AMB:=TREND.MB_RegistriLetti[176] ,
	UMID_ASS_EST:=TREND.MB_RegistriLetti[171]  ,
	UMID_ASS_AMB:= TREND.MB_RegistriLetti[178] ,
	UMID_ASS_MISC:=TREND.MB_RegistriLetti[179] ,
	UMID_ASS_CONDEN:=TREND.MB_RegistriLetti[180]  ,
	SET_COMP_T_AMB:=TREND.MB_RegistriLetti[168]  ,
	RITAR_SET_T_AMB:= TREND.MB_RegistriHoldingLetti[96],
	SET_T_MAND:= TREND.MB_RegistriHoldingLetti[88] ,
	SET_ANTIGELO:= TREND.MB_RegistriHoldingLetti[89] ,
	SET_UR_AMB:= TREND.MB_RegistriHoldingLetti[90],
	ISTERESI_UR_AMB:= TREND.MB_RegistriHoldingLetti[91] ,
	SET_F_ANTIG_AMB:= TREND.MB_RegistriHoldingLetti[92] ,
	SOGLIA_T_EST_VR:=  TREND.MB_RegistriHoldingLetti[93],
	MIN_AP_SERR_E_R:=  TREND.MB_RegistriHoldingLetti[94],
	MIN_AP_SERR_ESP:=  TREND.MB_RegistriHoldingLetti[95],
	RID_SET_T_RISC:=  TREND.MB_RegistriHoldingLetti[97],
	VENT_MAND:= TREND.MB_BitStato[114],
	VENT_RIPR:=TREND.MB_BitStato[115] ,
	P_UMIDIF:=TREND.MB_BitStato[116] ,
	VALV_B_FREDDA:=TREND.MB_BitStato[185] ,
	VALV_B_CALDA:=TREND.MB_BitStato[186] ,
	SERRANDE_ESP:= TREND.MB_BitStato[187],
	SERRAND_EST_RIC:= TREND.MB_BitStato[188],
	ABILITA:=TREND.MB_BitStatoCoil[21] ,
	STATO_VENT_M:=TREND.MB_BitStato[122] ,
	STATO_VENT_R:=TREND.MB_BitStato[123] ,
	FILTRO:=TREND.MB_BitStato[124] ,
	FLUSSO_VM:=TREND.MB_BitStato[125] ,
	FLUSSO_VR:= TREND.MB_BitStato[126],
	FILTRI_INTASATI:= TREND.MB_BitStato[134],
	ALL_VERIFICA_VM:=TREND.MB_BitStato[135] ,
	ALL_VERIFICA_VR:= TREND.MB_BitStato[136],
	ALL_V011_MANC_SPEGN:= TREND.MB_BitStato[137],
	ALL_V011_MANC_FUNZ:=TREND.MB_BitStato[138],
	ALL_V012_MANC_SPEGN:=TREND.MB_BitStato[139] ,
	ALL_V012_MANC_FUNZ:=TREND.MB_BitStato[140],
	cmd_DI_RUN:=THER03.RunCrono,
	cmd_DI_SetPoint:=THER03.SetPoint,
	UTA_CONTROL_MODE:=cmd_ControlMode_UTA03	);





	UTA04(
	UTA_ST:= TREND.MB_BitStatoCoil[22],     	(* ABILITA UTA6  *)
	UTA_CentrAL:=TREND.MB_BitStato[153] OR TREND.MB_BitStato[154],	 (* TRUE= Flusso , FALSE = No Flusso *)
	T_AMB:=TREND.MB_RegistriLetti[189] ,
	UR_AMB:=TREND.MB_RegistriLetti[190]  ,
	T_MISC:=TREND.MB_RegistriLetti[191]  ,
	UR_MISC:=TREND.MB_RegistriLetti[192]  ,
	T_MAND:=TREND.MB_RegistriLetti[193]  ,
	T_EST:=TREND.MB_RegistriLetti[199]  ,
	UR_EST:= TREND.MB_RegistriLetti[200] ,
	ENTALPIA_EST:=TREND.MB_RegistriLetti[203]  ,
	ENTALPIA_AMB:=TREND.MB_RegistriLetti[204] ,
	UMID_ASS_EST:=TREND.MB_RegistriLetti[205]  ,
	UMID_ASS_AMB:= TREND.MB_RegistriLetti[206] ,
	UMID_ASS_MISC:=TREND.MB_RegistriLetti[207] ,
	UMID_ASS_CONDEN:=TREND.MB_RegistriLetti[208]  ,
	SET_COMP_T_AMB:=TREND.MB_RegistriLetti[201]  ,
	RITAR_SET_T_AMB:= TREND.MB_RegistriHoldingLetti[98],
	SET_T_MAND:= TREND.MB_RegistriHoldingLetti[99] ,
	SET_ANTIGELO:= TREND.MB_RegistriHoldingLetti[100] ,
	SET_UR_AMB:= TREND.MB_RegistriHoldingLetti[101],
	ISTERESI_UR_AMB:= TREND.MB_RegistriHoldingLetti[102] ,
	SET_F_ANTIG_AMB:= TREND.MB_RegistriHoldingLetti[103] ,
	SOGLIA_T_EST_VR:=  TREND.MB_RegistriHoldingLetti[104],
	MIN_AP_SERR_E_R:=  TREND.MB_RegistriHoldingLetti[105],
	MIN_AP_SERR_ESP:=  TREND.MB_RegistriHoldingLetti[106],
	RID_SET_T_RISC:=  TREND.MB_RegistriHoldingLetti[107],
	VENT_MAND:= TREND.MB_BitStato[144],
	VENT_RIPR:=TREND.MB_BitStato[145] ,
	P_UMIDIF:=TREND.MB_BitStato[146] ,
	VALV_B_FREDDA:=TREND.MB_BitStato[215] ,
	VALV_B_CALDA:=TREND.MB_BitStato[216] ,
	SERRANDE_ESP:= TREND.MB_BitStato[217],
	SERRAND_EST_RIC:= TREND.MB_BitStato[218],
	ABILITA:=TREND.MB_BitStatoCoil[22] ,
	STATO_VENT_M:=TREND.MB_BitStato[150] ,
	STATO_VENT_R:=TREND.MB_BitStato[151] ,
	FILTRO:=TREND.MB_BitStato[152] ,
	FLUSSO_VM:=TREND.MB_BitStato[153] ,
	FLUSSO_VR:= TREND.MB_BitStato[154],
	FILTRI_INTASATI:= TREND.MB_BitStato[160],
	ALL_VERIFICA_VM:=TREND.MB_BitStato[161] ,
	ALL_VERIFICA_VR:= TREND.MB_BitStato[162],
	ALL_V011_MANC_SPEGN:= TREND.MB_BitStato[163],
	ALL_V011_MANC_FUNZ:=TREND.MB_BitStato[164],
	ALL_V012_MANC_SPEGN:=TREND.MB_BitStato[165] ,
	ALL_V012_MANC_FUNZ:=TREND.MB_BitStato[166],
	cmd_DI_RUN:=THER04.RunCrono,
	cmd_DI_SetPoint:=THER04.SetPoint,
	UTA_CONTROL_MODE:=cmd_ControlMode_UTA04);



	UTA05(
	UTA_ST:= TREND.MB_BitStatoCoil[23],     	(* V021 VENT.MAND.UTA2  *)
	UTA_CentrAL:=TREND.MB_BitStato[158] OR TREND.MB_BitStato[159],	 (* TRUE= Flusso , FALSE = No Flusso *)
	T_AMB:=TREND.MB_RegistriLetti[194] ,
	UR_AMB:=TREND.MB_RegistriLetti[195]  ,
	T_MISC:=TREND.MB_RegistriLetti[196]  ,
	UR_MISC:=TREND.MB_RegistriLetti[197]  ,
	T_MAND:=TREND.MB_RegistriLetti[198]  ,
	T_EST:=TREND.MB_RegistriLetti[199]  ,
	UR_EST:= TREND.MB_RegistriLetti[200] ,
	ENTALPIA_EST:=TREND.MB_RegistriLetti[203]  ,
	ENTALPIA_AMB:=TREND.MB_RegistriLetti[210] ,
	UMID_ASS_EST:=TREND.MB_RegistriLetti[205]  ,
	UMID_ASS_AMB:= TREND.MB_RegistriLetti[212] ,
	UMID_ASS_MISC:=TREND.MB_RegistriLetti[213] ,
	UMID_ASS_CONDEN:=TREND.MB_RegistriLetti[214]  ,
	SET_COMP_T_AMB:=TREND.MB_RegistriLetti[202]  ,
	RITAR_SET_T_AMB:= TREND.MB_RegistriHoldingLetti[116],
	SET_T_MAND:= TREND.MB_RegistriHoldingLetti[108] ,
	SET_ANTIGELO:= TREND.MB_RegistriHoldingLetti[109] ,
	SET_UR_AMB:= TREND.MB_RegistriHoldingLetti[110],
	ISTERESI_UR_AMB:= TREND.MB_RegistriHoldingLetti[111] ,
	SET_F_ANTIG_AMB:= TREND.MB_RegistriHoldingLetti[112] ,
	SOGLIA_T_EST_VR:=  TREND.MB_RegistriHoldingLetti[113],
	MIN_AP_SERR_E_R:=  TREND.MB_RegistriHoldingLetti[114],
	MIN_AP_SERR_ESP:=  TREND.MB_RegistriHoldingLetti[115],
	RID_SET_T_RISC:=  TREND.MB_RegistriHoldingLetti[117],
	VENT_MAND:= TREND.MB_BitStato[147],
	VENT_RIPR:=TREND.MB_BitStato[148] ,
	P_UMIDIF:=TREND.MB_BitStato[149] ,
	VALV_B_FREDDA:=TREND.MB_BitStato[219] ,
	VALV_B_CALDA:=TREND.MB_BitStato[220] ,
	SERRANDE_ESP:= TREND.MB_BitStato[221],
	SERRAND_EST_RIC:= TREND.MB_BitStato[222],
	ABILITA:=TREND.MB_BitStatoCoil[23] ,
	STATO_VENT_M:=TREND.MB_BitStato[155] ,
	STATO_VENT_R:=TREND.MB_BitStato[156] ,
	FILTRO:=TREND.MB_BitStato[157] ,
	FLUSSO_VM:=TREND.MB_BitStato[158] ,
	FLUSSO_VR:= TREND.MB_BitStato[159],
	FILTRI_INTASATI:= TREND.MB_BitStato[167],
	ALL_VERIFICA_VM:=TREND.MB_BitStato[168] ,
	ALL_VERIFICA_VR:= TREND.MB_BitStato[169],
	ALL_V011_MANC_SPEGN:= TREND.MB_BitStato[170],
	ALL_V011_MANC_FUNZ:=TREND.MB_BitStato[171],
	ALL_V012_MANC_SPEGN:=TREND.MB_BitStato[172] ,
	ALL_V012_MANC_FUNZ:=TREND.MB_BitStato[173],
	cmd_DI_RUN:=THER05.RunCrono,
	cmd_DI_SetPoint:=THER05.SetPoint,
	UTA_CONTROL_MODE:=cmd_ControlMode_UTA05);



	UTA06(
	UTA_ST:= TREND.MB_BitStatoCoil[1],     	(* V021 VENT.MAND.UTA2  *)
	UTA_CentrAL:=TREND.MB_BitStato[7] OR TREND.MB_BitStato[8],	 (* TRUE= Flusso , FALSE = No Flusso *)
	T_AMB:=TREND.MB_RegistriLetti[1] ,
	UR_AMB:=TREND.MB_RegistriLetti[2]  ,
	T_MISC:=TREND.MB_RegistriLetti[3]  ,
	UR_MISC:=TREND.MB_RegistriLetti[4]  ,
	T_MAND:=TREND.MB_RegistriLetti[5]  ,
	T_EST:=TREND.MB_RegistriLetti[6]  ,
	UR_EST:= TREND.MB_RegistriLetti[7] ,
	ENTALPIA_EST:=TREND.MB_RegistriLetti[8]  ,
	ENTALPIA_AMB:=TREND.MB_RegistriLetti[9] ,
	UMID_ASS_EST:=TREND.MB_RegistriLetti[10]  ,
	UMID_ASS_AMB:= TREND.MB_RegistriLetti[11] ,
	UMID_ASS_MISC:=TREND.MB_RegistriLetti[12] ,
	UMID_ASS_CONDEN:=TREND.MB_RegistriLetti[13]  ,
	SET_COMP_T_AMB:=TREND.MB_RegistriLetti[14]  ,
	RITAR_SET_T_AMB:= TREND.MB_RegistriHoldingLetti[15],
	SET_T_MAND:= TREND.MB_RegistriHoldingLetti[1] ,
	SET_ANTIGELO:= TREND.MB_RegistriHoldingLetti[2] ,
	SET_UR_AMB:= TREND.MB_RegistriHoldingLetti[3],
	ISTERESI_UR_AMB:= TREND.MB_RegistriHoldingLetti[4] ,
	SET_F_ANTIG_AMB:= TREND.MB_RegistriHoldingLetti[5] ,
	SOGLIA_T_EST_VR:=  TREND.MB_RegistriHoldingLetti[6],
	MIN_AP_SERR_E_R:=  TREND.MB_RegistriHoldingLetti[7],
	MIN_AP_SERR_ESP:=  TREND.MB_RegistriHoldingLetti[8],
	RID_SET_T_RISC:=  TREND.MB_RegistriHoldingLetti[9],
	VENT_MAND:= TREND.MB_BitStato[1],
	VENT_RIPR:=TREND.MB_BitStato[2] ,
	P_UMIDIF:=TREND.MB_BitStato[3] ,
	VALV_B_FREDDA:=TREND.MB_BitStato[16] ,
	VALV_B_CALDA:=TREND.MB_BitStato[17] ,
	SERRANDE_ESP:= TREND.MB_BitStato[18],
	SERRAND_EST_RIC:= TREND.MB_BitStato[19],
	ABILITA:=TREND.MB_BitStatoCoil[1] ,
	STATO_VENT_M:=TREND.MB_BitStato[4] ,
	STATO_VENT_R:=TREND.MB_BitStato[5] ,
	FILTRO:=TREND.MB_BitStato[6] ,
	FLUSSO_VM:=TREND.MB_BitStato[7] ,
	FLUSSO_VR:= TREND.MB_BitStato[8],
	FILTRI_INTASATI:= TREND.MB_BitStato[13],
	ALL_VERIFICA_VM:=TREND.MB_BitStato[14] ,
	ALL_VERIFICA_VR:= TREND.MB_BitStato[15],
	ALL_V011_MANC_SPEGN:= TREND.MB_BitStato[16],
	ALL_V011_MANC_FUNZ:=TREND.MB_BitStato[17],
	ALL_V012_MANC_SPEGN:=TREND.MB_BitStato[18] ,
	ALL_V012_MANC_FUNZ:=TREND.MB_BitStato[19],
	cmd_DI_RUN:=THER06.RunCrono,
	cmd_DI_SetPoint:=THER06.SetPoint,
	UTA_CONTROL_MODE:=cmd_ControlMode_UTA06);



	UTA07(
	UTA_ST:= TREND.MB_BitStatoCoil[2],     	(* ABILITA UTA6  *)
	UTA_CentrAL:=TREND.MB_BitStato[25] OR TREND.MB_BitStato[26],	 (* TRUE= Flusso , FALSE = No Flusso *)
	T_AMB:=TREND.MB_RegistriLetti[20] ,
	UR_AMB:=TREND.MB_RegistriLetti[21]  ,
	T_MISC:=TREND.MB_RegistriLetti[22]  ,
	UR_MISC:=TREND.MB_RegistriLetti[23]  ,
	T_MAND:=TREND.MB_RegistriLetti[24]  ,
	T_EST:=TREND.MB_RegistriLetti[36]  ,
	UR_EST:= TREND.MB_RegistriLetti[37] ,
	ENTALPIA_EST:=TREND.MB_RegistriLetti[29]  ,
	ENTALPIA_AMB:=TREND.MB_RegistriLetti[30] ,
	UMID_ASS_EST:=TREND.MB_RegistriLetti[31]  ,
	UMID_ASS_AMB:= TREND.MB_RegistriLetti[32] ,
	UMID_ASS_MISC:=TREND.MB_RegistriLetti[33] ,
	UMID_ASS_CONDEN:=TREND.MB_RegistriLetti[34]  ,
	SET_COMP_T_AMB:=TREND.MB_RegistriLetti[35]  ,
	RITAR_SET_T_AMB:= TREND.MB_RegistriHoldingLetti[10],
	SET_T_MAND:= TREND.MB_RegistriHoldingLetti[11] ,
	SET_ANTIGELO:= TREND.MB_RegistriHoldingLetti[12] ,
	SET_UR_AMB:= TREND.MB_RegistriHoldingLetti[13],
	ISTERESI_UR_AMB:= TREND.MB_RegistriHoldingLetti[14] ,
	SET_F_ANTIG_AMB:= TREND.MB_RegistriHoldingLetti[15] ,
	SOGLIA_T_EST_VR:=  TREND.MB_RegistriHoldingLetti[16],
	MIN_AP_SERR_E_R:=  TREND.MB_RegistriHoldingLetti[17],
	MIN_AP_SERR_ESP:=  TREND.MB_RegistriHoldingLetti[18],
	RID_SET_T_RISC:=  TREND.MB_RegistriHoldingLetti[19],
	VENT_MAND:= TREND.MB_BitStato[20],
	VENT_RIPR:=TREND.MB_BitStato[21] ,
	P_UMIDIF:=TREND.MB_BitStato[22] ,
	VALV_B_FREDDA:=TREND.MB_BitStato[38] ,
	VALV_B_CALDA:=TREND.MB_BitStato[39] ,
	SERRANDE_ESP:= TREND.MB_BitStato[40],
	SERRAND_EST_RIC:= TREND.MB_BitStato[41],
	ABILITA:=TREND.MB_BitStatoCoil[2] ,
	STATO_VENT_M:=TREND.MB_BitStato[358] ,
	STATO_VENT_R:=TREND.MB_BitStato[23] ,
	FILTRO:=TREND.MB_BitStato[24] ,
	FLUSSO_VM:=TREND.MB_BitStato[25] ,
	FLUSSO_VR:= TREND.MB_BitStato[26],
	FILTRI_INTASATI:= TREND.MB_BitStato[29],
	ALL_VERIFICA_VM:=TREND.MB_BitStato[30] ,
	ALL_VERIFICA_VR:= TREND.MB_BitStato[31],
	ALL_V011_MANC_SPEGN:= TREND.MB_BitStato[32],
	ALL_V011_MANC_FUNZ:=TREND.MB_BitStato[33],
	ALL_V012_MANC_SPEGN:=TREND.MB_BitStato[34] ,
	ALL_V012_MANC_FUNZ:=TREND.MB_BitStato[35],
	cmd_DI_RUN:=THER07.RunCrono,
	cmd_DI_SetPoint:=THER07.SetPoint,
	UTA_CONTROL_MODE:=cmd_ControlMode_UTA07);




	UTA08(
	UTA_ST:= TREND.MB_BitStatoCoil[10],     	(* V021 VENT.MAND.UTA2  *)
	UTA_CentrAL:=TREND.MB_BitStato[44] OR TREND.MB_BitStato[45],  	 (* TRUE= Flusso , FALSE = No Flusso *)
	T_AMB:=TREND.MB_RegistriLetti[46] ,
	UR_AMB:=TREND.MB_RegistriLetti[47]  ,
	T_MISC:=TREND.MB_RegistriLetti[48]  ,
	UR_MISC:=TREND.MB_RegistriLetti[49]  ,
	T_MAND:=TREND.MB_RegistriLetti[50]  ,
	T_EST:=TREND.MB_RegistriLetti[58]  ,
	UR_EST:= TREND.MB_RegistriLetti[59] ,
	ENTALPIA_EST:=TREND.MB_RegistriLetti[51]  ,
	ENTALPIA_AMB:=TREND.MB_RegistriLetti[52] ,
	UMID_ASS_EST:=TREND.MB_RegistriLetti[53]  ,
	UMID_ASS_AMB:= TREND.MB_RegistriLetti[54] ,
	UMID_ASS_MISC:=TREND.MB_RegistriLetti[55] ,
	UMID_ASS_CONDEN:=TREND.MB_RegistriLetti[56]  ,
	SET_COMP_T_AMB:=TREND.MB_RegistriLetti[57]  ,
	RITAR_SET_T_AMB:= TREND.MB_RegistriHoldingLetti[24],
	SET_T_MAND:= TREND.MB_RegistriHoldingLetti[25] ,
	SET_ANTIGELO:= TREND.MB_RegistriHoldingLetti[26] ,
	SET_UR_AMB:= TREND.MB_RegistriHoldingLetti[27],
	ISTERESI_UR_AMB:= TREND.MB_RegistriHoldingLetti[28] ,
	SET_F_ANTIG_AMB:= TREND.MB_RegistriHoldingLetti[29] ,
	SOGLIA_T_EST_VR:=  TREND.MB_RegistriHoldingLetti[30],
	MIN_AP_SERR_E_R:=  TREND.MB_RegistriHoldingLetti[31],
	MIN_AP_SERR_ESP:=  TREND.MB_RegistriHoldingLetti[32],
	RID_SET_T_RISC:=  TREND.MB_RegistriHoldingLetti[33],
	VENT_MAND:= TREND.MB_BitStato[38],
	VENT_RIPR:=TREND.MB_BitStato[39] ,
	P_UMIDIF:=TREND.MB_BitStato[40] ,
	VALV_B_FREDDA:=TREND.MB_BitStato[60] ,
	VALV_B_CALDA:=TREND.MB_BitStato[61] ,
	SERRANDE_ESP:= TREND.MB_BitStato[62],
	SERRAND_EST_RIC:= TREND.MB_BitStato[63],
	ABILITA:=TREND.MB_BitStatoCoil[10] ,
	STATO_VENT_M:=TREND.MB_BitStato[41] ,
	STATO_VENT_R:=TREND.MB_BitStato[42] ,
	FILTRO:=TREND.MB_BitStato[43] ,
	FLUSSO_VM:=TREND.MB_BitStato[44] ,
	FLUSSO_VR:= TREND.MB_BitStato[45],
	FILTRI_INTASATI:= TREND.MB_BitStato[48],
	ALL_VERIFICA_VM:=TREND.MB_BitStato[49] ,
	ALL_VERIFICA_VR:= TREND.MB_BitStato[50],
	ALL_V011_MANC_SPEGN:= TREND.MB_BitStato[51],
	ALL_V011_MANC_FUNZ:=TREND.MB_BitStato[52],
	ALL_V012_MANC_SPEGN:=TREND.MB_BitStato[53] ,
	ALL_V012_MANC_FUNZ:=TREND.MB_BitStato[54],
	cmd_DI_RUN:=THER08.RunCrono,
	cmd_DI_SetPoint:=THER08.SetPoint,
	UTA_CONTROL_MODE:=cmd_ControlMode_UTA08);





	UTA09(
	UTA_ST:= TREND.MB_BitStatoCoil[11],     	(* V021 VENT.MAND.UTA2  *)
	UTA_CentrAL:=TREND.MB_BitStato[61] OR TREND.MB_BitStato[62],	   (* TRUE= Flusso , FALSE = No Flusso *)
	T_AMB:=TREND.MB_RegistriLetti[65] ,
	UR_AMB:=TREND.MB_RegistriLetti[66]  ,
	T_MISC:=TREND.MB_RegistriLetti[67]  ,
	UR_MISC:=TREND.MB_RegistriLetti[68]  ,
	T_MAND:=TREND.MB_RegistriLetti[69]  ,
	T_EST:=TREND.MB_RegistriLetti[77]  ,
	UR_EST:= TREND.MB_RegistriLetti[78] ,
	ENTALPIA_EST:=TREND.MB_RegistriLetti[70]  ,
	ENTALPIA_AMB:=TREND.MB_RegistriLetti[71] ,
	UMID_ASS_EST:=TREND.MB_RegistriLetti[72]  ,
	UMID_ASS_AMB:= TREND.MB_RegistriLetti[73] ,
	UMID_ASS_MISC:=TREND.MB_RegistriLetti[74] ,
	UMID_ASS_CONDEN:=TREND.MB_RegistriLetti[75]  ,
	SET_COMP_T_AMB:=TREND.MB_RegistriLetti[76]  ,
	RITAR_SET_T_AMB:= TREND.MB_RegistriHoldingLetti[34],
	SET_T_MAND:= TREND.MB_RegistriHoldingLetti[35] ,
	SET_ANTIGELO:= TREND.MB_RegistriHoldingLetti[36] ,
	SET_UR_AMB:= TREND.MB_RegistriHoldingLetti[37],
	ISTERESI_UR_AMB:= TREND.MB_RegistriHoldingLetti[38] ,
	SET_F_ANTIG_AMB:= TREND.MB_RegistriHoldingLetti[39] ,
	SOGLIA_T_EST_VR:=  TREND.MB_RegistriHoldingLetti[40],
	MIN_AP_SERR_E_R:=  TREND.MB_RegistriHoldingLetti[41],
	MIN_AP_SERR_ESP:=  TREND.MB_RegistriHoldingLetti[42],
	RID_SET_T_RISC:=  TREND.MB_RegistriHoldingLetti[43],
	VENT_MAND:= TREND.MB_BitStato[55],
	VENT_RIPR:=TREND.MB_BitStato[56] ,
	P_UMIDIF:=TREND.MB_BitStato[57] ,
	VALV_B_FREDDA:=TREND.MB_BitStato[79] ,
	VALV_B_CALDA:=TREND.MB_BitStato[80] ,
	SERRANDE_ESP:= TREND.MB_BitStato[81],
	SERRAND_EST_RIC:= TREND.MB_BitStato[82],
	ABILITA:=TREND.MB_BitStatoCoil[11] ,
	STATO_VENT_M:=TREND.MB_BitStato[58] ,
	STATO_VENT_R:=TREND.MB_BitStato[59] ,
	FILTRO:=TREND.MB_BitStato[60] ,
	FLUSSO_VM:=TREND.MB_BitStato[61] ,
	FLUSSO_VR:= TREND.MB_BitStato[62],
	FILTRI_INTASATI:= TREND.MB_BitStato[65],
	ALL_VERIFICA_VM:=TREND.MB_BitStato[66] ,
	ALL_VERIFICA_VR:= TREND.MB_BitStato[67],
	ALL_V011_MANC_SPEGN:= TREND.MB_BitStato[68],
	ALL_V011_MANC_FUNZ:=TREND.MB_BitStato[69],
	ALL_V012_MANC_SPEGN:=TREND.MB_BitStato[70] ,
	ALL_V012_MANC_FUNZ:=TREND.MB_BitStato[71],
	cmd_DI_RUN:=THER09.RunCrono,
	cmd_DI_SetPoint:=THER09.SetPoint,
	UTA_CONTROL_MODE:=cmd_ControlMode_UTA09);


	UTA10(
	UTA_ST:= TREND.MB_BitStatoCoil[65],     	(* ABILITA UTA6  *)
	UTA_CentrAL:=TREND.MB_BitStato[338] OR TREND.MB_BitStato[339],	 (* TRUE= Flusso , FALSE = No Flusso *)
	T_AMB:=TREND.MB_RegistriLetti[266] ,
	UR_AMB:=TREND.MB_RegistriLetti[267]  ,
	T_MISC:=TREND.MB_RegistriLetti[268]  ,
	UR_MISC:=TREND.MB_RegistriLetti[269]  ,
	T_MAND:=TREND.MB_RegistriLetti[270]  ,
	T_EST:=TREND.MB_RegistriLetti[279]  ,
	UR_EST:= TREND.MB_RegistriLetti[280] ,
	ENTALPIA_EST:=TREND.MB_RegistriLetti[272]  ,
	ENTALPIA_AMB:=TREND.MB_RegistriLetti[273] ,
	UMID_ASS_EST:=TREND.MB_RegistriLetti[274]  ,
	UMID_ASS_AMB:= TREND.MB_RegistriLetti[275] ,
	UMID_ASS_MISC:=TREND.MB_RegistriLetti[276] ,
	UMID_ASS_CONDEN:=TREND.MB_RegistriLetti[277]  ,
	SET_COMP_T_AMB:=TREND.MB_RegistriLetti[278]  ,
	RITAR_SET_T_AMB:= TREND.MB_RegistriLetti[271],
	SET_T_MAND:= TREND.MB_RegistriHoldingLetti[160] ,
	SET_ANTIGELO:= TREND.MB_RegistriHoldingLetti[161] ,
	SET_UR_AMB:= TREND.MB_RegistriHoldingLetti[162],
	ISTERESI_UR_AMB:= TREND.MB_RegistriHoldingLetti[163] ,
	SET_F_ANTIG_AMB:= TREND.MB_RegistriHoldingLetti[164] ,
	SOGLIA_T_EST_VR:=  TREND.MB_RegistriHoldingLetti[165],
	MIN_AP_SERR_E_R:=  TREND.MB_RegistriHoldingLetti[166],
	MIN_AP_SERR_ESP:=  TREND.MB_RegistriHoldingLetti[167],
	RID_SET_T_RISC:=  TREND.MB_RegistriHoldingLetti[168],
	VENT_MAND:= TREND.MB_BitStato[330],
	VENT_RIPR:=TREND.MB_BitStato[331] ,
	P_UMIDIF:=TREND.MB_BitStato[332] ,
	VALV_B_FREDDA:=TREND.MB_BitStato[281] ,
	VALV_B_CALDA:=TREND.MB_BitStato[282] ,
	SERRANDE_ESP:= TREND.MB_BitStato[283],
	SERRAND_EST_RIC:= TREND.MB_BitStato[284],
	ABILITA:=TREND.MB_BitStatoCoil[65] ,
	STATO_VENT_M:=TREND.MB_BitStato[335] ,
	STATO_VENT_R:=TREND.MB_BitStato[336] ,
	FILTRO:=TREND.MB_BitStato[337] ,
	FLUSSO_VM:=TREND.MB_BitStato[338] ,
	FLUSSO_VR:= TREND.MB_BitStato[339],
	FILTRI_INTASATI:= TREND.MB_BitStato[343],
	ALL_VERIFICA_VM:=TREND.MB_BitStato[344] ,
	ALL_VERIFICA_VR:= TREND.MB_BitStato[345],
	ALL_V011_MANC_SPEGN:= TREND.MB_BitStato[346],
	ALL_V011_MANC_FUNZ:=TREND.MB_BitStato[347],
	ALL_V012_MANC_SPEGN:=TREND.MB_BitStato[348] ,
	ALL_V012_MANC_FUNZ:=TREND.MB_BitStato[349],
	cmd_DI_RUN:=THER10.RunCrono,
	cmd_DI_SetPoint:=THER10.SetPoint,
	UTA_CONTROL_MODE:=cmd_ControlMode_UTA10);




(*	UTA11( 	UTA_ST:= TREND.MB_BitStatoCoil[111],     	(* V021 VENT.MAND.UTA2  *)
			UTA_CentrAL:=TREND.MB_BitStato[100] OR TREND.MB_BitStato[101],	(* ALLARME FLUSSO  *)
		 ); *)
	UTA12(
	UTA_ST:= TREND.MB_BitStatoCoil[14],     	(* V021 VENT.MAND.UTA2  *)
	UTA_CentrAL:=FALSE,	 (* TRUE= Flusso , FALSE = No Flusso *)
	T_AMB:=TREND.MB_RegistriLetti[97] ,
	UR_AMB:=-9999  ,
	T_MISC:=-9999  ,
	UR_MISC:=-9999  ,
	T_MAND:=TREND.MB_RegistriLetti[98]  ,
	T_EST:=TREND.MB_RegistriLetti[108]  ,
	UR_EST:= -9999 ,
	ENTALPIA_EST:=-9999  ,
	ENTALPIA_AMB:=-9999 ,
	UMID_ASS_EST:=-9999 ,
	UMID_ASS_AMB:= -9999 ,
	UMID_ASS_MISC:=-9999 ,
	UMID_ASS_CONDEN:=-9999 ,
	SET_COMP_T_AMB:=TREND.MB_RegistriLetti[103]  ,
	RITAR_SET_T_AMB:= TREND.MB_RegistriHoldingLetti[52] ,
	SET_T_MAND:= TREND.MB_RegistriHoldingLetti[53] ,
	SET_ANTIGELO:= TREND.MB_RegistriHoldingLetti[54] ,
	SET_UR_AMB:= -9999,
	ISTERESI_UR_AMB:= -9999 ,
	SET_F_ANTIG_AMB:= -9999 ,
	SOGLIA_T_EST_VR:=  -9999,
	MIN_AP_SERR_E_R:=  -9999,
	MIN_AP_SERR_ESP:=  -9999,
	RID_SET_T_RISC:=  TREND.MB_RegistriHoldingLetti[56],
	VENT_MAND:= TREND.MB_BitStato[77],
	VENT_RIPR:=0 ,
	P_UMIDIF:= 0 ,
	VALV_B_FREDDA:=TREND.MB_BitStato[109] ,
	VALV_B_CALDA:=TREND.MB_BitStato[110] ,
	SERRANDE_ESP:=0,
	SERRAND_EST_RIC:= TREND.MB_BitStato[76],
	ABILITA:=TREND.MB_BitStatoCoil[14] ,
	STATO_VENT_M:=TREND.MB_BitStato[81],
	STATO_VENT_R:=0 ,
	FILTRO:=TREND.MB_BitStato[78] ,
	FLUSSO_VM:=TREND.MB_BitStato[79] ,
	FLUSSO_VR:= 0,
	FILTRI_INTASATI:= TREND.MB_BitStato[82],
	ALL_VERIFICA_VM:=TREND.MB_BitStato[83] ,
	ALL_VERIFICA_VR:=0,
	ALL_V011_MANC_SPEGN:= TREND.MB_BitStato[84],
	ALL_V011_MANC_FUNZ:=TREND.MB_BitStato[85],
	ALL_V012_MANC_SPEGN:=0 ,
	ALL_V012_MANC_FUNZ:=0,
	cmd_DI_RUN:=THER12.RunCrono,
	cmd_DI_SetPoint:=THER12.SetPoint,
	UTA_CONTROL_MODE:=cmd_ControlMode_UTA12);




	UTA13(
	UTA_ST:= TREND.MB_BitStatoCoil[18],     	(* ABILITA UTA6  *)
	UTA_CentrAL:=TREND.MB_BitStato[79] ,	 (* TRUE= Flusso , FALSE = No Flusso *)
	T_AMB:=TREND.MB_RegistriLetti[121] ,
	UR_AMB:=-9999  ,
	T_MISC:=-9999  ,
	UR_MISC:=-9999  ,
	T_MAND:=TREND.MB_RegistriLetti[122]  ,
	T_EST:=TREND.MB_RegistriLetti[131]  ,
	UR_EST:= -9999 ,
	ENTALPIA_EST:=-9999  ,
	ENTALPIA_AMB:=-9999 ,
	UMID_ASS_EST:=-9999 ,
	UMID_ASS_AMB:= -9999 ,
	UMID_ASS_MISC:=-9999 ,
	UMID_ASS_CONDEN:=-9999 ,
	SET_COMP_T_AMB:=TREND.MB_RegistriLetti[126]  ,
	RITAR_SET_T_AMB:= TREND.MB_RegistriHoldingLetti[63] ,
	SET_T_MAND:= TREND.MB_RegistriHoldingLetti[64] ,
	SET_ANTIGELO:= TREND.MB_RegistriHoldingLetti[65] ,
	SET_UR_AMB:= -9999,
	ISTERESI_UR_AMB:= -9999 ,
	SET_F_ANTIG_AMB:= -9999 ,
	SOGLIA_T_EST_VR:=  -9999,
	MIN_AP_SERR_E_R:=  -9999,
	MIN_AP_SERR_ESP:=  -9999,
	RID_SET_T_RISC:=  TREND.MB_RegistriHoldingLetti[67],
	VENT_MAND:= TREND.MB_BitStato[90],
	VENT_RIPR:=0 ,
	P_UMIDIF:= 0 ,
	VALV_B_FREDDA:=TREND.MB_BitStato[132] ,
	VALV_B_CALDA:=TREND.MB_BitStato[133] ,
	SERRANDE_ESP:=0,
	SERRAND_EST_RIC:= TREND.MB_BitStato[89],
	ABILITA:=TREND.MB_BitStatoCoil[18] ,
	STATO_VENT_M:=TREND.MB_BitStato[94],
	STATO_VENT_R:=0 ,
	FILTRO:=TREND.MB_BitStato[91] ,
	FLUSSO_VM:=TREND.MB_BitStato[92] ,
	FLUSSO_VR:= 0,
	FILTRI_INTASATI:= TREND.MB_BitStato[95],
	ALL_VERIFICA_VM:=TREND.MB_BitStato[96] ,
	ALL_VERIFICA_VR:=0,
	ALL_V011_MANC_SPEGN:= TREND.MB_BitStato[97],
	ALL_V011_MANC_FUNZ:=TREND.MB_BitStato[98],
	ALL_V012_MANC_SPEGN:=0 ,
	ALL_V012_MANC_FUNZ:=0,
	cmd_DI_RUN:=THER13.RunCrono,
	cmd_DI_SetPoint:=THER13.SetPoint,
	UTA_CONTROL_MODE:=cmd_ControlMode_UTA13);




	MODB02();


	ANZ01(ModBus:=MODB02);	(* Generale  *)
	ANZ02(ModBus:=MODB02);	(* QE. Uffici - QU  *)
	ANZ03(ModBus:=MODB02);	(* Gruppo frigo 1  *)
	ANZ04(ModBus:=MODB02);	(* Gruppo frigo 2  *)
	ANZ05(ModBus:=MODB02);	(* Q.E. UTA 1-5  *)
	ANZ06(ModBus:=MODB02);	(* Linee UTA (n.3 - una per fase) *)
	ANZ07(ModBus:=MODB02);	(* Linee UTA (n.3 - una per fase) *)
	ANZ08(ModBus:=MODB02);	(* Linee UTA (n.2 - una per fase) *)


	NodoDaInterrogareANZ:=LIMIT(1,NodoDaInterrogareANZ,9);
	IF NodoDaInterrogareANZ>8 THEN NodoDaInterrogareANZ:=1;END_IF;



	MODB03();

	ZTHL01(MODBUS:=MODB03);
	ZTHL02(MODBUS:=MODB03);
	ZTHL03(MODBUS:=MODB03);
	ZTHL04(MODBUS:=MODB03);
	ZTHL05(MODBUS:=MODB03);
	ZTHL06(MODBUS:=MODB03);

	COOV01(MODBUS:=MODB03);
	COOV02(MODBUS:=MODB03);
	COOV03(MODBUS:=MODB03);
	COOV04(MODBUS:=MODB03);
	COOV05(MODBUS:=MODB03);
	COOV06(MODBUS:=MODB03);

	GATEWAY(MODBUS:=MODB03);


	NodoDaInterrogareMB2:=LIMIT(1,NodoDaInterrogareMB2,14);
	IF NodoDaInterrogareMB2>13 THEN NodoDaInterrogareMB2:=1;END_IF;


	(* ModBus *)
	MODB04();

(*	CHI01.Temperatura:=T_AMB;
	CHI01.SetPointManuale:= SEL(THER07.SetPoint=0,THER07.SetPoint,200); *)

	CHIAERMEC01(ModBus:=MODB04, CLIM:=CHI01_Clima,
	 	AbilitaSetPointManuale:=NOT (THER07.SetPoint=1000));
	CHIAERMEC02(ModBus:=MODB04, CLIM:=CHI02_Clima,
	 	AbilitaSetPointManuale:=NOT (THER07.SetPoint=1000));

	NodoDaInterrogareChiller:=LIMIT(1,NodoDaInterrogareChiller,3);
	IF NodoDaInterrogareChiller>2 THEN NodoDaInterrogareChiller:=1;END_IF;








END_IF

(*==============================*)
(*== System cycle operations ===*)
(*==============================*)
(* Execute TCP processes *)
Logger_Proc();
Remote_Proc();

(* Update user led *)
(* USRLED_Update(); *)

(* *)








(* Execute Cron Editor commands *)
CronEd();
END_PROGRAM
ACTION Main_Stm:
CASE Sys.Status OF

	S_STARTUP:
		Sys.Status:=S_INIT_RTC;

	S_INIT_RTC:
		(* Check RTC and update from network *)
		RTC_Update();
		(* Check time *)
		IF Sys.Time_Year>2000 THEN
			Sys.Status:=S_INIT_VAR;
		END_IF

	S_INIT_VAR:
		LogEv(EL_Wrn,EO_SYS,0,1,CONCAT('System_startup_v',WORD_TO_STRING(Plant_SW_VER)));
		Sys.Status:=S_RUNNING;

	S_RUNNING:
		Timer1(IN:=NOT Timer1.Q,PT:=T#50ms);
		IF Timer1.Q THEN
			(* Update meters *)

			(* Update system checks *)
			SYS_Proc();
		END_IF

		Timer2(IN:=NOT Timer2.Q,PT:=T#500ms);
		IF Timer2.Q THEN
			(* Read current date/time *)
			RTC_Update();

			(* Thermostats *)
			THER01(Temperature:=100);
			THER02(Temperature:=100);
			THER03(Temperature:=100);
			THER04(Temperature:=100);
			THER05(Temperature:=100);
			THER06(Temperature:=100);
		    	THER07(Temperature:=100);
		    	THER08(Temperature:=100);
		    	THER09(Temperature:=100);
		    	THER10(Temperature:=100);
		    	THER12(Temperature:=100);
		    	THER13(Temperature:=100);

			(* Test toggle *)
			(*IF TEST1 THEN TEST1:=FALSE; ELSE TEST1:=TRUE; END_IF*)
		END_IF

		Timer3(IN:=NOT Timer3.Q,PT:=T#5m);

		R_TRIG_CHIAERMEC01_ScriviDato(clk:=CHIAERMEC01.ScriviDato);
		R_TRIG_CHIAERMEC02_ScriviDato(clk:=CHIAERMEC02.ScriviDato);
		R_TRIG_TREND_ScriviDato(clk:=TREND.ScriviDato);

		IF  R_TRIG_CHIAERMEC01_ScriviDato.q OR R_TRIG_CHIAERMEC02_ScriviDato.Q OR R_TRIG_TREND_ScriviDato.Q THEN
			aggiornalogdaModBus:=TRUE;
		END_IF

		tonaggiornaLogdaModBus(in:=aggiornalogdaModBus,pt:=t#5s);

		R_TrigAggiornaLog(clk:=Timer3.Q OR AggiornaLog OR tonaggiornaLogdaModBus.Q OR RichiestaLogDaRemoto);

		IF  R_TrigAggiornaLog.Q  THEN
			aggiornalogdaModBus:=FALSE;
			(* Trig logger *)
			(* LogTrig(); *)
			EseguiLog:=10;
			(* Execute temporary CSV logger *)
			(*CSV_Log();*)
		END_IF

		allarme:= (
				THER01.Status_Log=2 OR
				THER02.Status_Log=2 OR
				THER03.Status_Log=2 OR
				THER04.Status_Log=2 OR
				THER05.Status_Log=2 OR
				THER06.Status_Log=2 OR
			     	THER07.Status_Log=2 OR
			     	THER08.Status_Log=2 OR
			     	THER09.Status_Log=2 OR
			     	THER10.Status_Log=2 OR
			     	THER12.Status_Log=2 OR
			     	THER13.Status_Log=2 OR
				UTA01.Status_Log=2 OR
				UTA02.Status_Log=2 OR
				UTA03.Status_Log=2 OR
				UTA04.Status_Log=2 OR
				UTA05.Status_Log=2 OR
				UTA06.Status_Log=2 OR
				UTA07.Status_Log=2 OR
				UTA08.Status_Log=2 OR
				UTA09.Status_Log=2 OR
				UTA10.Status_Log=2 OR

				ANZ01.Status_Log=2 OR
				ANZ02.Status_Log=2 OR
				ANZ03.Status_Log=2 OR
				ANZ04.Status_Log=2 OR
				ANZ05.Status_Log=2 OR
				ANZ06.Status_Log=2 OR
				ANZ07.Status_Log=2 OR
				ANZ08.Status_Log=2 OR

				ZTHL01.Status_Log=2 OR
				ZTHL02.Status_Log=2 OR
				ZTHL03.Status_Log=2 OR
				ZTHL04.Status_Log=2 OR
				ZTHL05.Status_Log=2 OR
				ZTHL06.Status_Log=2 OR

				COOV01.Status_Log=2 OR
				COOV02.Status_Log=2 OR
				COOV03.Status_Log=2 OR
				COOV04.Status_Log=2 OR
				COOV05.Status_Log=2 OR
				COOV06.Status_Log=2 OR

				CHIAERMEC01.Status_Log=2 OR
				CHIAERMEC02.Status_Log=2 OR
				TREND.Status_Log=2
				);

		warning:= (
				THER01.Status_Log=1 OR
				THER02.Status_Log=1 OR
				THER03.Status_Log=1 OR
				THER04.Status_Log=1 OR
				THER05.Status_Log=1 OR
				THER06.Status_Log=1 OR
			      THER07.Status_Log=1 OR
			      THER08.Status_Log=1 OR
			      THER09.Status_Log=1 OR
			      THER10.Status_Log=1 OR
			      THER12.Status_Log=1 OR
			      THER13.Status_Log=1 OR
				UTA01.Status_Log=1 OR
				UTA02.Status_Log=1 OR
				UTA03.Status_Log=1 OR
				UTA04.Status_Log=1 OR
				UTA05.Status_Log=1 OR
				UTA06.Status_Log=1 OR
				UTA07.Status_Log=1 OR
				UTA08.Status_Log=1 OR
				UTA09.Status_Log=1 OR
				UTA10.Status_Log=1 OR

				ANZ01.Status_Log=1 OR
				ANZ02.Status_Log=1 OR
				ANZ03.Status_Log=1 OR
				ANZ04.Status_Log=1 OR
				ANZ05.Status_Log=1 OR
				ANZ06.Status_Log=1 OR
				ANZ07.Status_Log=1 OR
				ANZ08.Status_Log=1 OR

				ZTHL01.Status_Log=1 OR
				ZTHL02.Status_Log=1 OR
				ZTHL03.Status_Log=1 OR
				ZTHL04.Status_Log=1 OR
				ZTHL05.Status_Log=1 OR
				ZTHL06.Status_Log=1 OR

				COOV01.Status_Log=1 OR
				COOV02.Status_Log=1 OR
				COOV03.Status_Log=1 OR
				COOV04.Status_Log=1 OR
				COOV05.Status_Log=1 OR
				COOV06.Status_Log=1 OR

				CHIAERMEC01.Status_Log=1 OR
				CHIAERMEC02.Status_Log=1 OR
				TREND.Status_Log=1
				);

		Lamp( Allarme:=	(allarme),
			  Warning:=  (warning),
			  SistemaInAllarme => Sys.Alarm,
			 SistemaWarning => Sys.Warning,
			 AllarmeLampada=>LAMP_AL
			 );


		CASE Eseguilog OF

			10 : 	Ton_pausaTrig(IN:=FALSE , PT:=t#5s , Q=> , ET=> );

					Logger_Head();

					THER01.AddLogData();
					THER02.AddLogData();
					THER03.AddLogData();
					THER04.AddLogData();
					THER05.AddLogData();
					THER06.AddLogData();
					THER07.AddLogData();
					THER08.AddLogData();
					THER09.AddLogData();
					THER10.AddLogData();
					THER12.AddLogData();
					THER13.AddLogData();

					UTA01.AddLogData();
					UTA02.AddLogData();
					UTA03.AddLogData();
					UTA04.AddLogData();
					UTA05.AddLogData();
					UTA06.AddLogData();
					UTA07.AddLogData();
					UTA08.AddLogData();
					UTA09.AddLogData();
					UTA10.AddLogData();
					(*UTA11.AddLogData();*)
					UTA12.AddLogData();
					UTA13.AddLogData();


					ANZ01.AddLogData(ModBus:=MODB02);
					ANZ02.AddLogData(ModBus:=MODB02);
					ANZ03.AddLogData(ModBus:=MODB02);
					ANZ04.AddLogData(ModBus:=MODB02);
					ANZ05.AddLogData(ModBus:=MODB02);
					ANZ06.AddLogData(ModBus:=MODB02);
					ANZ07.AddLogData(ModBus:=MODB02);
					ANZ08.AddLogData(ModBus:=MODB02);

					Logger_Send();

					s1:='';
					s1:=CONCAT(s1,REPLACE(Sys.Time_LogString,'T',1,11));
					Sys.LastLogs_Dat[Sys.LastLogs_Idx]:=s1;
					Sys.LastLogs_Msg[Sys.LastLogs_Idx]:='invio_Primo_Log';
					Sys.LastLogs_Idx:=Sys.LastLogs_Idx+1;
					IF Sys.LastLogs_Idx>5 THEN Sys.LastLogs_Idx:=0; END_IF
					RichiestaLogDaRemoto:=FALSE;
					EseguiLog:=20;
				20: Ton_pausaTrig(IN:=TRUE , PT:=t#10s , Q=> , ET=> );
					IF Ton_pausaTrig.Q THEN
						EseguiLog:=30;
					END_IF

				30 : Ton_pausaTrig(IN:=FALSE , PT:=t#2s , Q=> , ET=> );
					Logger_Head();

					ZTHL01.AddLogData(ModBus:=MODB03);
					ZTHL02.AddLogData(ModBus:=MODB03);
					ZTHL03.AddLogData(ModBus:=MODB03);
					ZTHL04.AddLogData(ModBus:=MODB03);
					ZTHL05.AddLogData(ModBus:=MODB03);
					ZTHL06.AddLogData(ModBus:=MODB03);

					COOV01.AddLogData(ModBus:=MODB03);
					COOV02.AddLogData(ModBus:=MODB03);
					COOV03.AddLogData(ModBus:=MODB03);
					COOV04.AddLogData(ModBus:=MODB03);
					COOV05.AddLogData(ModBus:=MODB03);
					COOV06.AddLogData(ModBus:=MODB03);

					CHIAERMEC01.AddLogData(ModBus:=MODB04,CLIM:=CHI01_Clima);
					CHIAERMEC02.AddLogData(ModBus:=MODB04,CLIM:=CHI02_Clima);
					TREND.AddLogData(ModBus:=MODB01);

					Logger_Send();
					s1:='';
					s1:=CONCAT(s1,REPLACE(Sys.Time_LogString,'T',1,11));
					Sys.LastLogs_Dat[Sys.LastLogs_Idx]:=s1;
					Sys.LastLogs_Msg[Sys.LastLogs_Idx]:='invio_Secondo_Log';
					Sys.LastLogs_Idx:=Sys.LastLogs_Idx+1;
					IF Sys.LastLogs_Idx>5 THEN Sys.LastLogs_Idx:=0; END_IF


						EseguiLog:=200;

				200: RichiestaLogDaRemoto:=FALSE;

		END_CASE

	S_SHUTDOWN:
		(* Stop sistema *)
		Sys.Status:=S_STARTUP;

	S_HALT:
		(* Aspetta uscita manuale *)
		Sys.Status:=S_STARTUP;

ELSE
	Sys.Status:=S_STARTUP;
END_CASE;
END_ACTION

(* POU TCP_Logger/Logger_Proc, ST *)
PROGRAM Logger_Proc
VAR
	c1:         	TCPCLIENT;

	Open:	    	BOOL;
	IpAddr:			DWORD;
	InetAddr:		DWORD;
	Connected:  	BOOL;
	Error:      	DINT;
	TxTrig:     	BOOL;
	RxData:			ARRAY [0..MAX_RECEIVE_TCP_CLIENT] OF BYTE;
	RxLen:			DINT;

	Retry:			BYTE;	(* Counter for connection retries *)
	Recovered:		BYTE;	(* Counter for recovered unsent messages *)

	i:				DINT;
	pos:			DWORD;
	hFile:			DWORD;

END_VAR
(*=== State machine ===*)
CASE Logger.Status OF

	S_Logger_UNKNOWN:
		(* Startup *)
		Logger.SendReq:=FALSE;
		Open:=FALSE;
		Logger.Status:=S_Logger_IDLE;

	S_Logger_IDLE:
		(* Wait request *)
		IF Logger.SendReq THEN
			(* Resolve server name or use static IP *)
			IF LEN(Logger_SERVER)=0 THEN
				InetAddr:=SysSockInetAddr(Logger_IP);
			ELSE
				IpAddr:=SysSockGetHostByName(ADR(Logger_SERVER));
				DWORDSWAP(pIn:=ADR(IpAddr), pOut:=ADR(InetAddr));
			END_IF
			TxTrig:=FALSE;
			RxLen:=0;
			(* Open connection *)
			Open:=TRUE;
			Logger.Status:=S_Logger_WAITCONN;
		END_IF

	S_Logger_WAITCONN:
		(* Wait connection *)
		IF Connected THEN
			(* Send data *)
			TxTrig:=TRUE;
			Logger.Status:=S_Logger_WAITTX;
		END_IF
		IF Error>0 THEN
			Open:=FALSE;
			Logger.Status:=S_Logger_ERROR;
		END_IF

	S_Logger_WAITTX:
		(* Wait transmission *)
		IF NOT TxTrig THEN
			Logger.Status:=S_Logger_WAITRESP;
		END_IF
		IF Error>0 THEN
			Open:=FALSE;
			Logger.Status:=S_Logger_ERROR;
		END_IF

	S_Logger_WAITRESP:
		(* Wait response *)
		IF Connected=FALSE (* OR TIMEOUT!! *) THEN
			Open:=FALSE;
			(* Check response *)
			IF RxLen>=4 AND CHKSTRING(pString:=ADR(RxData), pPattern:=ADR(Logger_CHECK)) THEN
				Logger.SendReq:=FALSE;
				Retry:=0;
				(* Check unsent messages to flush *)
				IF Recovered<Logger_RecoverMsgs THEN
					MsgChk();
					IF Logger.SendReq=TRUE THEN
						Recovered:=Recovered+1;
					ELSE
						Recovered:=0;
					END_IF
				ELSE
					Recovered:=0;
				END_IF
				Logger.Status:=S_Logger_IDLE;
			ELSE
				Logger.Status:=S_Logger_ERROR;
			END_IF
		END_IF

	S_Logger_ERROR:
		(* Connection error or send failure *)
		Retry:=Retry+1;
		IF Retry>Logger_ConnRetries THEN
			(* Save message as unsent *)
			MsgSave();
			Logger.SendReq:=FALSE;
			Retry:=0;
		END_IF
		Logger.Status:=S_Logger_IDLE;

ELSE
	Logger.Status:=S_Logger_UNKNOWN;
END_CASE


(*=== Execute client lib ===*)
c1(
	xOpenConnection			:= Open,
	dwInetAddr 				:= InetAddr,
	wPortNumber				:= Logger_PORT,
	ptSendData				:= ADR(Logger.SendData),
	diSendCount				:= Logger.SendLen,
	tConnectWatchdogTime	:= t#10s,
	xStartSend				:= TxTrig,
	aReceiveBuffer			:= RxData,
	diReceiveCount			:= RxLen,
	xConnected				=> Connected,
	diError					=> Error
);

(*=== Process Rx data ===*)
(*IF RxLen>0 THEN
	RxLen:=0;
END_IF*)
END_PROGRAM
ACTION MsgChk:
(* Open index file *)
hFile:=SysFileOpen(Logger_IndexFile,'r');
IF hFile=0 THEN
	RETURN;
END_IF
(* Search oldest message to recover *)
SysFileSetPos(hFile,Logger.LastIdxPos);
Logger.SendLen:=0;
REPEAT
	SysFileRead(hFile, ADR(Logger.SendIdx), SIZEOF(Logger.SendIdx));
	pos:=SysFileGetPos(hFile);
	SysFileRead(hFile, ADR(Logger.SendLen), SIZEOF(Logger.SendLen));
UNTIL
	SysFileEOF(hFile) OR Logger.SendLen<>0
END_REPEAT
SysFileClose(hFile);
(* Delete index file when all messages are recovered *)
IF Logger.SendLen=0 THEN
	Logger.LastIdxPos:=0;
	SysFileDelete(Logger_IndexFile);
	RETURN;
END_IF
(* Recover message data *)
hFile:=SysFileOpen(Logger_DataFile,'r');
IF hFile<>0 THEN
	SysFileSetPos(hFile,Logger.SendIdx);
	SysFileRead(hFile,ADR(Logger.SendData),Logger.SendLen);
	Logger.SendReq:=TRUE;
	SysFileClose(hFile);
END_IF
(* Clear index entry *)
hFile:=SysFileOpen(Logger_IndexFile,'rw');
IF hFile<>0 THEN
	SysFileSetPos(hFile,pos);
	i:=0;
	SysFileWrite(hFile, ADR(i), 4);
	Logger.LastIdxPos:=SysFileGetPos(hFile);
	SysFileClose(hFile);
END_IF
END_ACTION
ACTION MsgSave:
(* Add log position in recovery indexes *)
hFile:=SysFileOpen(Logger_IndexFile,'a');
SysFileWrite(hFile, ADR(Logger.SendIdx), SIZEOF(Logger.SendIdx));
SysFileWrite(hFile, ADR(Logger.SendLen), SIZEOF(Logger.SendLen));
SysFileClose(hFile);
END_ACTION

(* POU Utils Functions/TCPCLIENT, ST *)
FUNCTION_BLOCK TCPCLIENT
(***********************************************************************************************************	*)
(* Version: 1.3b                        			          													*)
(* Date: 28.10.2014                   				          							            			*)
(***********************************************************************************************************	*)
(* WAGO Kontakttechnik GmbH Hansastr. 27 32423 Minden(Westf.)													*)
(* Tel. +0049 571/887-0 Fax. +0049 571/887-0																	*)
(* Author: VB																									*)
(***********************************************************************************************************	*)
(*Description:	A TCP client to read and write data with additional connection watchdog							*)
(*History:																										*)
(*Version 1.3b: 28.10.2014: Use DWORD address for IP (Andrea Ravasio)											*)
(*Version 1.3: 11.02.2011: Changes according to 750-880/881											 			*)
(*Version 1.2: 29.08.2007 Bugfix TCP Client																		*)
(*Version 1.1: 15.01.2007 Changes according to FW11																*)
(*Version 1.0: 09.03.2006 Release																				*)
(***********************************************************************************************************	*)
VAR CONSTANT
	STATE_CREATE     				 : BYTE:= 0;
	STATE_OPEN     					 : BYTE:= 1;
	STATE_IOCTL    					 : BYTE:= 2;
	STATE_CONNECT     				 : BYTE:= 10;
	STATE_TX       					 : BYTE:= 20;
	STATE_RX       					 : BYTE:= 30;
	STATE_CLOSE    					 : BYTE:= 40;
	STATE_ERROR_TRAP			     : BYTE:= 200;
END_VAR

VAR_INPUT
	xOpenConnection					: BOOL;
	dwInetAddr						: DWORD; (* <== Use SysSockInetAddr() value or
													swapped bytes order of SysSockGetHostByName() value *)
	wPortNumber						: WORD;
	ptSendData						: POINTER TO ARRAY[0..MAX_SEND_TCP_CLIENT] OF BYTE;
	diSendCount						: DINT;
	tConnectWatchdogTime		    : TIME := t#10s;
END_VAR
VAR_OUTPUT
	xConnected						: BOOL;
	diError 						: DINT := 0;
END_VAR
(* ErrorCodes -----------------------------------------
	16#8001 => No socket descriptor available 
	16#8002 => SysSockSend returns -1 
	16#8003 => Socket was "gracefully closed" 
	16#8004 => switching to none blocking mode fails
	16#8005 => SysSockClose() returns FALSE 
    16#8006 => SysSockConnect() fails
    16#8007 => SysSockSend() fails
	16#8008 => error state machine 
	16#8009 => timeout while waiting for data from server 
------------------------------------------------------------*)
VAR_IN_OUT
	xStartSend							: BOOL;
	aReceiveBuffer						: ARRAY [0..MAX_RECEIVE_TCP_CLIENT] OF BYTE;
	diReceiveCount						: DINT;
END_VAR
VAR
	m_State								: BYTE := 0;
	m_ReceiveBuffer						: ARRAY [0..MAX_RECEIVE_TCP_CLIENT_SOCKET] OF BYTE;
	m_Socket							: DINT;
	m_AddressInfo						: SOCKADDRESS;
	m_BytesReceived						: DINT;
	m_diReturn							: DINT;
	m_xReturn							: BOOL;
	m_IoCtlParameter  					: DINT := 1; (* IOCTL-Parameter for non-blocking mode of sockets *)
	i									: INT;
	T_Connect							: TON;
	m_count								: DINT;
	diOption							: DINT := 1;
	m_Blocking   						: DINT := 0;
END_VAR
IF xOpenConnection THEN
	(* State maschine *)
	CASE  m_State OF

	(* -------------------------------------------------------------------------*)
	STATE_CREATE:
			(* create socket descriptor*)
			m_Socket := SysSockCreate(diAddressFamily	:= SOCKET_AF_INET,
													 diType		:= SOCKET_STREAM,
													 diProtocol := SOCKET_IPPROTO_TCP);
			IF m_Socket >= 0 THEN
			(*Set Push-Bit*)
				IF ADR(%MW0)=16#30000000  OR ADR(%MW0)=16#20000000 THEN (*841 or 881*)
					SysSockSetOption(
						diSocket:=m_Socket,
						diLevel:=6,
						diOption:=SOCKET_TCP_NODELAY,
						pOptionValue:=ADR(diOption),
						diOptionLength:=SIZEOF(diOption));
				ELSE
						;
				END_IF
				m_State := STATE_IOCTL; (* succesful *)
			ELSE
				diError := 16#8001;  (* no socket descriptor available *)
				m_State := STATE_ERROR_TRAP;
			END_IF

	(* -------------------------------------------------------------------------*)
	STATE_IOCTL: (* change  socket mode  to none blocking *)
		m_diReturn := SysSockIoctl( m_Socket, SOCKET_FIONBIO, ADR(m_IoCtlParameter));
		IF m_diReturn <> 0 THEN
			m_AddressInfo.sin_family := SOCKET_AF_INET;
			m_AddressInfo.sin_port := SysSockNtohs(wPortNumber);
			m_AddressInfo.sin_addr := dwInetAddr;
			m_State := STATE_CONNECT;
		ELSE
			diError := 16#8004;  (* switching to none blocking mode fails *)
			m_State := STATE_ERROR_TRAP;
		END_IF


	(* -------------------------------------------------------------------------*)
	STATE_CONNECT: (* connect with server *)
		T_Connect(IN:=TRUE , PT:=tConnectWatchdogTime);(*activate watchdog for establishing connection to a server*)
		m_xReturn := SysSockConnect ( m_Socket, ADR(m_AddressInfo),  SIZEOF(m_AddressInfo));
		IF m_xReturn THEN (* succesful *)
			IF xStartSend THEN
				m_State := STATE_TX;(*transmit data*)
			ELSE
				m_State := STATE_RX;(*wait for data from server*)
			END_IF
			xConnected:=TRUE;
			T_Connect(IN:=FALSE);
		ELSE
			IF T_Connect.Q THEN
				diError := 16#8006;  (* connect fails *)
				xConnected:=FALSE;
				T_Connect(IN:=FALSE);
				m_State := STATE_ERROR_TRAP;
				SysSockClose( m_Socket);
			ELSE
				m_State := STATE_CONNECT;(*client still  tries to set up connection*)
			END_IF
		END_IF


	STATE_TX:	 (* send TCP-message *)
		m_diReturn := SysSockSend(diSocket := m_Socket,
								  pbyBuffer := ADR(ptSendData^[0]),
								  diBufferSize := diSendCount-m_count,
								  diFlags := 0);

		CASE m_diReturn OF
		-1:	(* ERROR *)
			T_Connect(IN:=TRUE , PT:=CONNECT_WATCHDOG_TIME);(*activate watchdog to check communication*)
			IF t_Connect.Q THEN
				diError := 16#8007;
				T_Connect(IN:=FALSE);
				m_State:=STATE_CLOSE;
			END_IF
		0: (* socket was "gracefully closed" *)
			m_State := STATE_CLOSE;
			diError := 16#8003;
		ELSE (* succesful *)
			m_count:=m_count+m_diReturn;
			IF m_count>=diSendCount THEN
				diError := 16#0000;
				m_State := STATE_RX;
				m_count:=0;
				xStartSend:=FALSE;
			END_IF
			T_Connect(IN:=FALSE);
		END_CASE

	(* -------------------------------------------------------------------------*)
	STATE_RX: (* process receive data *)
			m_BytesReceived := SysSockRecv(	diSocket 	:= m_Socket,
										pbyBuffer 	:= ADR(m_ReceiveBuffer),		(* Address of receive buffer *)
										diBufferSize:= SIZEOF(m_ReceiveBuffer),
										diFlags		:= 0);

			CASE m_BytesReceived OF
			-1:	(* No data available or error occured *)
				T_Connect(IN:=TRUE , PT:=tConnectWatchdogTime);(*activate watchdog to check communication*)
				IF t_Connect.Q THEN
					diError:=16#8009;
					T_Connect(IN:=FALSE);
					m_State:=STATE_CLOSE;
				END_IF
				IF xStartSend THEN
					m_State:=STATE_TX	;(* WAIT IN THIS STATE  and check for arriving data or new send command*)
				END_IF;
			0: (* socket was "gracefully closed"  *)
				m_State:=STATE_CLOSE;
				diError := 16#8003;
			ELSE (* succesful *)
				diError := 16#0000;
				T_Connect(IN:=FALSE);
				(* Copy received data into receive buffer *)
				FOR i:= 0 TO DINT_TO_INT(m_BytesReceived	)-1 DO
					aReceiveBuffer[diReceiveCount]:= m_ReceiveBuffer[i];
					diReceiveCount:=(diReceiveCount+1) MOD SIZEOF(aReceiveBuffer);
				END_FOR

			END_CASE

	(* -------------------------------------------------------------------------*)
	STATE_CLOSE : (* close socket *)
		IF ADR(%MW0)=16#30000000  OR ADR(%MW0)=16#20000000 THEN (*841 or 881*)
			;
		ELSE
			SysSockShutdown(m_Socket, 0);;(*870*)
		END_IF
		m_xReturn := SysSockClose( m_Socket);
		m_Socket := -1;
		m_State := 0; (* succesful *)
		xConnected:=FALSE;
		T_Connect(IN:=FALSE);
	(* -------------------------------------------------------------------------*)
	STATE_ERROR_TRAP: (* error handling *)
		xConnected:=FALSE;

	ELSE  (* Bad FSM code trap  *)
			m_State:= STATE_ERROR_TRAP;
			diError:= 16#8008;
	END_CASE

ELSE(*close connection*)
	IF m_Socket >= 0 THEN
		IF ADR(%MW0)=16#30000000  OR ADR(%MW0)=16#20000000 THEN (*841 or 881*)
			;
		ELSE
			SysSockShutdown(m_Socket, 0);;(*870*)
		END_IF
		SysSockClose( m_Socket);
	END_IF
	m_Socket := -1;
	diError := 16#0000;
	m_State := STATE_CREATE;
	xConnected:=FALSE;
	T_Connect(IN:=FALSE);
END_IF
END_FUNCTION_BLOCK

(* POU Utils Functions/DWORDSWAP, ST *)
FUNCTION DWORDSWAP:BOOL
VAR_INPUT
	pIn:POINTER TO ARRAY[1..4] OF BYTE;
	pOut:POINTER TO ARRAY[1..4] OF BYTE;
END_VAR
VAR
END_VAR
pOut^[1]:=pIn^[4];
pOut^[2]:=pIn^[3];
pOut^[3]:=pIn^[2];
pOut^[4]:=pIn^[1];
END_FUNCTION

(* POU Utils Functions/CHKSTRING, ST *)
FUNCTION CHKSTRING : BOOL
VAR_INPUT
	pString: POINTER TO BYTE;
	pPattern: POINTER TO BYTE;
END_VAR
VAR
END_VAR
CHKSTRING:=TRUE;
WHILE pPattern^<>0 AND CHKSTRING DO
	IF pPattern^<>pString^ THEN CHKSTRING:=FALSE; END_IF
	pString:=pString+1;
	pPattern:=pPattern+1;
END_WHILE
END_FUNCTION

(* POU TCP_Remote/Remote_Proc, ST *)
PROGRAM Remote_Proc
VAR
	s1:         	TCPSERVER;
	Enable: 		BOOL;
	Connected: 		BOOL;
	Error: 			DINT;

	TxData:			ARRAY [0..MAX_SEND_TCP_SERVER] OF BYTE;
	TxLen:			DINT;
	TxTrig:			BOOL;

	RxData:			ARRAY [0..MAX_RECEIVE_TCP_SERVER] OF BYTE;
	RxLen:			DINT;

	Status:			DINT;

	(* Command interpreter *)

	Cmd_Buf:		ARRAY [0..MAX_RECEIVE_TCP_SERVER] OF BYTE;
	Cmd_Buf_U16:	POINTER TO WORD;
	Cmd_Buf_INT:	POINTER TO INT;
	Cmd_BufLen:		WORD;
	Cmd_St:			WORD;

	Cmd_Obj:		WORD;
	Cmd_ObjIdx:		WORD;
	Cmd_C:			WORD;
	Cmd_R:			WORD;
	Cmd_CLen:		WORD;
	Cmd_RLen:		WORD;

	i : WORD;
	j : INT;
	s2 : STRING;

		(* per aggiornare la data e l'ora *)
	SetAnno: INT;
	SetMese: INT;
	SetGiorno: INT;
	SetOra: INT;
	SetMinuti: INT;
	SetSecondi: INT;




END_VAR
(*=== State machine ===*)
CASE Status OF
	0: (* Startup *)
		TxLen:=0; TxTrig:=FALSE;
		RxLen:=0;
		Enable:=TRUE;
		Status:=1;

	1: (* Wait incoming connection *)
		IF Connected THEN
			(* Log access *)(*
			LogEv(EL_Log,EO_VPN,1,5,'Remote');*)
			(* Send welcome message *)(*
			ADDSTRING(pTxData:=ADR(TxData), pString:=ADR(Remote_WELCOME), TxLen:=TxLen);
			TxTrig:=TRUE;*)
			(* Reset vars *)
			Cmd_BufLen:=0;
			Cmd_St:=0;
			Status:=2;
		END_IF
		IF Error>1 THEN
			Enable:=FALSE;
			Status:=0;
		END_IF

	2: (* Wait command *)
		IF RxLen>0 THEN
			(*=== Interpreter start ===*)
			IF Cmd_BufLen+(RxLen/2)>=MAX_RECEIVE_TCP_SERVER THEN
				(* ERROR *)
				Cmd_BufLen:=0;
			ELSE
				i:=HEXTORAW(pString:=ADR(RxData), StringLen:=DINT_TO_WORD(RxLen), pData:=ADR(Cmd_Buf[Cmd_BufLen]));
				Cmd_BufLen:=Cmd_BufLen+i;
			END_IF
			IF Cmd_BufLen>=8 THEN
				Cmd_Buf_U16:=ADR(Cmd_Buf[6]);
				IF Cmd_BufLen>=(8+Cmd_Buf_U16^) THEN
					Cmd_CLen:=Cmd_Buf_U16^;
					Cmd_Buf_U16:=ADR(Cmd_Buf[0]); Cmd_Obj:=Cmd_Buf_U16^;
					Cmd_Buf_U16:=ADR(Cmd_Buf[2]); Cmd_ObjIdx:=Cmd_Buf_U16^;
					Cmd_Buf_U16:=ADR(Cmd_Buf[4]); Cmd_C:=Cmd_Buf_U16^;
					(* Log command *)(*
					s2:='RCmd_';		s2:=CONCAT(s2,WORD_TO_STRING(Cmd_Obj));
					s2:=CONCAT(s2,'_'); s2:=CONCAT(s2,WORD_TO_STRING(Cmd_ObjIdx));
					s2:=CONCAT(s2,'_'); s2:=CONCAT(s2,WORD_TO_STRING(Cmd_C));
					s2:=CONCAT(s2,'_');	s2:=CONCAT(s2,WORD_TO_STRING(Cmd_CLen));
					LogEv(EL_Log,EO_VPN,1,6,s2);*)
					(* Execute command *)
					Command();
					Cmd_BufLen:=0;
				END_IF
			END_IF
			(*=== Interpreter end ===*)
			RxLen:=0;
		END_IF
		IF NOT Connected THEN
			Status:=0;
		END_IF

ELSE
	Status:=0;
END_CASE


(*=== Execute server lib ===*)
s1(
	xEnable				:= Enable,
	wPortNumber			:= Remote_PORT,
	tServerTimeOut		:= t#15m,
	ptSendData			:= ADR(TxData),
	diSendCount			:= TxLen,
	xStartSend			:= TxTrig,
	aReceiveBuffer		:= RxData,
	diReceiveCount		:= RxLen,
	xClientConnected	=> Connected,
	diError				=> Error
);
END_PROGRAM
ACTION cmd_CHIAERMEC:
(* Check index *)

IF Cmd_ObjIdx<1 OR Cmd_ObjIdx>2 THEN
	Cmd_R:=2;
	RETURN;
END_IF

(* Process command *)
CASE Cmd_C OF

	1: (* GET CLIMATIC *)
		Cmd_RLen:=20;
		FOR i:=0 TO 4 DO
			j:=DINT_TO_INT(CHI01_Clima.Points[i].X);
			TxLen:=TxLen+RAWTOHEX(ADR(j),2,ADR(TxData[TxLen]));
			j:=DINT_TO_INT(CHI01_Clima.Points[i].Y);
			TxLen:=TxLen+RAWTOHEX(ADR(j),2,ADR(TxData[TxLen]));
		END_FOR

	2: (* SET CLIMATIC *)
		IF Cmd_CLen<>20 THEN
			Cmd_R:=4;
		ELSE
			FOR i:=0 TO 4 DO
				Cmd_Buf_INT:=ADR(Cmd_Buf[8+4*i]); j:=Cmd_Buf_INT^;
				CHI01_Clima.Points[i].X:=(j);(*INT_TO_DINT(j); *)
				Cmd_Buf_INT:=ADR(Cmd_Buf[10+4*i]); j:=Cmd_Buf_INT^;
				CHI01_Clima.Points[i].Y:=(j); (*INT_TO_DINT(j); *)
			END_FOR
		END_IF


	3:	(* Force On *)
		CASE Cmd_ObjIdx OF

			1:	CHIAERMEC01.RUN_REQ := TRUE;
			2:	CHIAERMEC02.RUN_REQ := TRUE;

		END_CASE

	4:	(* Force Off *)
		CASE Cmd_ObjIdx OF

			1:	CHIAERMEC01.STOP_REQ := TRUE;
			2:	CHIAERMEC02.STOP_REQ := TRUE;

		END_CASE

	5:	(* Release force *)
		CASE Cmd_ObjIdx OF

			1:	CHIAERMEC01.RUN_REQ	:= FALSE;
				CHIAERMEC01.STOP_REQ := FALSE;
			2:	CHIAERMEC02.RUN_REQ	:= FALSE;
				CHIAERMEC02.STOP_REQ := FALSE;

		END_CASE

	6: (* SET Tempi delay On Off   *)
		CASE Cmd_ObjIdx OF
			1:	Cmd_Buf_U16:=ADR(Cmd_Buf[8]);
				CHIAERMEC01.OnDelay := DWORD_TO_TIME((Cmd_Buf_U16^)*60*1000); 			(* Delay ON*)
				Cmd_Buf_U16:=ADR(Cmd_Buf[10]);
				CHIAERMEC01.OffDelay := DWORD_TO_TIME((Cmd_Buf_U16^)*60*1000);			(* Delay OFF *)

		END_CASE


	7: (* GET Tempi delay On Off  *)
		Cmd_RLen:=4;
			CASE Cmd_ObjIdx OF


			1:	j:=DWORD_TO_WORD(TIME_TO_DWORD((CHIAERMEC01.OnDelay)/60/1000));
				TxLen:=TxLen+RAWTOHEX(ADR(j),2,ADR(TxData[TxLen]));
				j:=DWORD_TO_WORD(TIME_TO_DWORD((CHIAERMEC01.OffDelay)/60/1000));
				TxLen:=TxLen+RAWTOHEX(ADR(j),2,ADR(TxData[TxLen]));
			2:	j:=DWORD_TO_WORD(TIME_TO_DWORD((CHIAERMEC01.OnDelay)/60/1000));
				TxLen:=TxLen+RAWTOHEX(ADR(j),2,ADR(TxData[TxLen]));
				j:=DWORD_TO_WORD(TIME_TO_DWORD((CHIAERMEC01.OffDelay)/60/1000));
				TxLen:=TxLen+RAWTOHEX(ADR(j),2,ADR(TxData[TxLen]));

			END_CASE

	8: (* SET Comandi  *)
		CASE Cmd_ObjIdx OF
			1:	Cmd_Buf_U16:=ADR(Cmd_Buf[8]);
				CHIAERMEC01.ChillerAbilitato := DWORD_TO_BOOL(Cmd_Buf_U16^); 	(* Chiller Abilitato 0=Disabilitato   1=abilitato *)
				Cmd_Buf_U16:=ADR(Cmd_Buf[10]);
				CHIAERMEC01.ImpMB_ResetFrigo := DWORD_TO_BOOL(Cmd_Buf_U16^); (* Comando reset sicurezze1=RESET  *)
				Cmd_Buf_U16:=ADR(Cmd_Buf[12]);
				CHIAERMEC01.ImpMB_LocRem := DWORD_TO_BOOL(Cmd_Buf_U16^); 	(* Comando locale/remoto (toggle)0=LOCALE   1=REMOTO  *)

				CHIAERMEC01.fWriteAttivazioneComandi:= TRUE;		(* da abilitare mettendo a true - abilitazione scrittura variabile Modbus *)
				CHIAERMEC01.Refresh_Now := TRUE;

		END_CASE



	9: (* GET Comandi  *)
		Cmd_RLen:=6;
			CASE Cmd_ObjIdx OF


			1:	j:=BOOL_TO_INT(CHIAERMEC01.ChillerAbilitato);
				TxLen:=TxLen+RAWTOHEX(ADR(j),2,ADR(TxData[TxLen]));
				j:=BOOL_TO_INT(CHIAERMEC01.MB_BitStato[2]);				(* Comando reset sicurezze1=RESET  *)
				TxLen:=TxLen+RAWTOHEX(ADR(j),2,ADR(TxData[TxLen]));
				j:=BOOL_TO_INT(CHIAERMEC01.MB_BitStato[3]);				(* Comando locale/remoto (toggle)0=LOCALE   1=REMOTO  *)
				TxLen:=TxLen+RAWTOHEX(ADR(j),2,ADR(TxData[TxLen]));
			2:	j:=BOOL_TO_INT(CHIAERMEC01.ChillerAbilitato);
				TxLen:=TxLen+RAWTOHEX(ADR(j),2,ADR(TxData[TxLen]));
				j:=BOOL_TO_INT(CHIAERMEC01.MB_BitStato[2]);				(* Comando reset sicurezze1=RESET  *)
				TxLen:=TxLen+RAWTOHEX(ADR(j),2,ADR(TxData[TxLen]));
				j:=BOOL_TO_INT(CHIAERMEC01.MB_BitStato[3]);				(* Comando locale/remoto (toggle)0=LOCALE   1=REMOTO  *)
				TxLen:=TxLen+RAWTOHEX(ADR(j),2,ADR(TxData[TxLen]));
       	END_CASE



	10: (* SET Comandi  *)
		CASE Cmd_ObjIdx OF
			1:	Cmd_Buf_U16:=ADR(Cmd_Buf[8]);
				CHIAERMEC01.ScriviCoil := DWORD_TO_BOOL(Cmd_Buf_U16^); 	(* 0 write on register - 1 write on coil *)
				Cmd_Buf_U16:=ADR(Cmd_Buf[10]);
				CHIAERMEC01.IndirizzoDaScrivere :=(Cmd_Buf_U16^); 		(* Address of the register / coil.  *)
				Cmd_Buf_U16:=ADR(Cmd_Buf[12]);
				CHIAERMEC01.DatoDaScrivere := (Cmd_Buf_U16^); 			(* The value to be written.  *)

				CHIAERMEC01.ScriviDato:= TRUE;							(* da abilitare mettendo a true - abilitazione scrittura variabile Modbus *)
				CHIAERMEC01.Refresh_Now := TRUE;

			2:	Cmd_Buf_U16:=ADR(Cmd_Buf[8]);
				CHIAERMEC02.ScriviCoil := DWORD_TO_BOOL(Cmd_Buf_U16^); 	(* 0 write on register - 1 write on coil *)
				Cmd_Buf_U16:=ADR(Cmd_Buf[10]);
				CHIAERMEC02.IndirizzoDaScrivere :=(Cmd_Buf_U16^); 		(* Address of the register / coil.  *)
				Cmd_Buf_U16:=ADR(Cmd_Buf[12]);
				CHIAERMEC02.DatoDaScrivere := (Cmd_Buf_U16^); 			(* The value to be written.  *)

				CHIAERMEC02.ScriviDato:= TRUE;							(* da abilitare mettendo a true - abilitazione scrittura variabile Modbus *)
				CHIAERMEC02.Refresh_Now := TRUE;
		END_CASE






ELSE
	Cmd_R:=3;
END_CASE
END_ACTION
ACTION Cmd_CRON:
(* Check index *)
IF Cmd_ObjIdx<1 OR Cmd_ObjIdx>13 THEN
	Cmd_R:=2;
	RETURN;
END_IF

(* Process command *)
CASE Cmd_C OF

	1: (* GET PROFILE *)
		IF Cmd_CLen<>3 THEN
			Cmd_R:=4;
		ELSE
			(* Load profile *)
			CronEd.CN_Sel:=WORD_TO_BYTE(Cmd_ObjIdx);
			Cmd_Buf_U16:=ADR(Cmd_Buf[8]);
			CronEd.CN_YSel:=Cmd_Buf_U16^;
			IF Cmd_Buf[10]<=10 THEN
				CronEd.PR_Sel:=Cmd_Buf[10];
				CronEd.PR_Load_Exe();
				(* Response data *)
				Cmd_RLen:=192;
				TxLen:=TxLen+RAWTOHEX(ADR(CronEd.PR.Setpoint),192,ADR(TxData[TxLen]));
			ELSE
				Cmd_R:=6;
			END_IF
		END_IF

	2: (* SET PROFILE *)
		IF Cmd_CLen<>(3+192) THEN
			Cmd_R:=4;
		ELSE
			(* Save profile *)
			CronEd.CN_Sel:=WORD_TO_BYTE(Cmd_ObjIdx);
			Cmd_Buf_U16:=ADR(Cmd_Buf[8]);
			CronEd.CN_YSel:=Cmd_Buf_U16^;
			IF Cmd_Buf[10]<=10 THEN
				CronEd.PR_Sel:=Cmd_Buf[10];
				MEMCPY(ADR(Cmd_Buf[11]),ADR(CronEd.PR.Setpoint),192);
				CronEd.PR_Save_Exe_Multi(); (* updated by DB - for saving profiles in eventually existing multiple crono files *)
			ELSE
				Cmd_R:=6;
			END_IF
		END_IF

	5: (* GET CALENDAR MONTH *)
		IF Cmd_CLen<>3 THEN
			Cmd_R:=4;
		ELSE
			(* Load calendar *)
			CronEd.CN_Sel:=WORD_TO_BYTE(Cmd_ObjIdx);
			Cmd_Buf_U16:=ADR(Cmd_Buf[8]);
			CronEd.CN_YSel:=Cmd_Buf_U16^;
			IF Cmd_Buf[10]>=1 AND Cmd_Buf[10]<=12 THEN
				CronEd.CA_Sel:=Cmd_Buf[10];
				CronEd.CA_Load_Exe();
				(* Response data *)
				Cmd_RLen:=32;
				TxLen:=TxLen+RAWTOHEX(ADR(CronEd.CA.Profile),32,ADR(TxData[TxLen]));
			ELSE
				Cmd_R:=6;
			END_IF
		END_IF

	6: (* SET CALENDAR MONTH *)
		IF Cmd_CLen<>(3+32) THEN
			Cmd_R:=4;
		ELSE
			(* Save calendar *)
			CronEd.CN_Sel:=WORD_TO_BYTE(Cmd_ObjIdx);
			Cmd_Buf_U16:=ADR(Cmd_Buf[8]);
			CronEd.CN_YSel:=Cmd_Buf_U16^;
			IF Cmd_Buf[10]>=1 AND Cmd_Buf[10]<=12 THEN
				CronEd.CA_Sel:=Cmd_Buf[10];
				MEMCPY(ADR(Cmd_Buf[11]),ADR(CronEd.CA.Profile),32);
				CronEd.CA_Save_Exe();
			ELSE
				Cmd_R:=6;
			END_IF
		END_IF




	9: (* CRON RESTART *)
		CASE Cmd_ObjIdx OF
			1: THER01.InitOK:=FALSE;
			2: THER02.InitOK:=FALSE;
			3: THER03.InitOK:=FALSE;
			4: THER04.InitOK:=FALSE;
			5: THER05.InitOK:=FALSE;
			6: THER06.InitOK:=FALSE;
			7: THER07.InitOK:=FALSE;
			8: THER08.InitOK:=FALSE;
			9: THER09.InitOK:=FALSE;
			10: THER10.InitOK:=FALSE;
			12: THER12.InitOK:=FALSE;
			13: THER13.InitOK:=FALSE;


		END_CASE

	10: (* SET Isteresi  *)
		CASE Cmd_ObjIdx OF
			1:	Cmd_Buf_U16:=ADR(Cmd_Buf[8]);
				THER01.Histeresys := Cmd_Buf_U16^; 			(* Isteresi*)
			2:	Cmd_Buf_U16:=ADR(Cmd_Buf[8]);
				THER02.Histeresys := Cmd_Buf_U16^; 			(* Isteresi*)
			3:	Cmd_Buf_U16:=ADR(Cmd_Buf[8]);
				THER03.Histeresys := Cmd_Buf_U16^; 			(* Isteresi*)
			4:	Cmd_Buf_U16:=ADR(Cmd_Buf[8]);
				THER04.Histeresys := Cmd_Buf_U16^; 			(* Isteresi*)
			5:	Cmd_Buf_U16:=ADR(Cmd_Buf[8]);
				THER05.Histeresys := Cmd_Buf_U16^; 			(* Isteresi*)
			6:	Cmd_Buf_U16:=ADR(Cmd_Buf[8]);
				THER06.Histeresys := Cmd_Buf_U16^; 			(* Isteresi*)
			7:	Cmd_Buf_U16:=ADR(Cmd_Buf[8]);
				THER07.Histeresys := Cmd_Buf_U16^; 			(* Isteresi*)
			8:	Cmd_Buf_U16:=ADR(Cmd_Buf[8]);
				THER08.Histeresys := Cmd_Buf_U16^; 			(* Isteresi*)
			9:	Cmd_Buf_U16:=ADR(Cmd_Buf[8]);
				THER09.Histeresys := Cmd_Buf_U16^; 			(* Isteresi*)
			10:	Cmd_Buf_U16:=ADR(Cmd_Buf[8]);
				THER10.Histeresys := Cmd_Buf_U16^; 			(* Isteresi*)
			12:	Cmd_Buf_U16:=ADR(Cmd_Buf[8]);
				THER12.Histeresys := Cmd_Buf_U16^; 			(* Isteresi*)
			13:	Cmd_Buf_U16:=ADR(Cmd_Buf[8]);
				THER13.Histeresys := Cmd_Buf_U16^; 			(* Isteresi*)



		END_CASE

	11: (* GET isteresi *)
		Cmd_RLen:=2;
		CASE Cmd_ObjIdx OF


			1: j:=(THER01.Histeresys);
				TxLen:=TxLen+RAWTOHEX(ADR(j),2,ADR(TxData[TxLen]));
			2: j:=(THER02.Histeresys);
				TxLen:=TxLen+RAWTOHEX(ADR(j),2,ADR(TxData[TxLen]));
			3: j:=(THER03.Histeresys);
				TxLen:=TxLen+RAWTOHEX(ADR(j),2,ADR(TxData[TxLen]));
			4: j:=(THER04.Histeresys);
				TxLen:=TxLen+RAWTOHEX(ADR(j),2,ADR(TxData[TxLen]));
			5: j:=(THER05.Histeresys);
				TxLen:=TxLen+RAWTOHEX(ADR(j),2,ADR(TxData[TxLen]));
			6: j:=(THER06.Histeresys);
				TxLen:=TxLen+RAWTOHEX(ADR(j),2,ADR(TxData[TxLen]));
			7: j:=(THER07.Histeresys);
				TxLen:=TxLen+RAWTOHEX(ADR(j),2,ADR(TxData[TxLen]));
			8: j:=(THER08.Histeresys);
				TxLen:=TxLen+RAWTOHEX(ADR(j),2,ADR(TxData[TxLen]));
			9: j:=(THER09.Histeresys);
				TxLen:=TxLen+RAWTOHEX(ADR(j),2,ADR(TxData[TxLen]));
			10: j:=(THER10.Histeresys);
				TxLen:=TxLen+RAWTOHEX(ADR(j),2,ADR(TxData[TxLen]));
			12: j:=(THER12.Histeresys);
				TxLen:=TxLen+RAWTOHEX(ADR(j),2,ADR(TxData[TxLen]));
			13: j:=(THER13.Histeresys);
				TxLen:=TxLen+RAWTOHEX(ADR(j),2,ADR(TxData[TxLen]));

		END_CASE
ELSE
	Cmd_R:=3;
END_CASE
END_ACTION
ACTION Cmd_Pool:
(* Check index *)
IF Cmd_ObjIdx<>1 THEN
	Cmd_R:=2;
	RETURN;
END_IF

(* Process command *)
CASE Cmd_C OF


	10: (* SET Comandi  *)
		CASE Cmd_ObjIdx OF
			1:	Cmd_Buf_U16:=ADR(Cmd_Buf[8]);
				TREND.ScriviCoil := DWORD_TO_BOOL(Cmd_Buf_U16^); 	(* 0 write on register - 1 write on coil *)
				Cmd_Buf_U16:=ADR(Cmd_Buf[10]);
				TREND.IndirizzoDaScrivere :=(Cmd_Buf_U16^); 		(* Address of the register / coil.  *)
				Cmd_Buf_U16:=ADR(Cmd_Buf[12]);
				TREND.DatoDaScrivere := (Cmd_Buf_U16^); 			(* The value to be written.  *)

				TREND.ScriviDato:= TRUE;		 					(* da abilitare mettendo a true - abilitazione scrittura variabile Modbus *)
				TREND.Refresh_Now := TRUE;

			END_CASE






ELSE
	Cmd_R:=3;
END_CASE
END_ACTION
ACTION Cmd_SYS:
(* Check index *)
IF Cmd_ObjIdx<>0 THEN
	Cmd_R:=2;
	RETURN;
END_IF

(* Process command *)
CASE Cmd_C OF

	0: (* ECHO *)
		IF Cmd_CLen<>0 THEN
			TxLen:=0;
		END_IF

	1: (* LOG REQUEST *)
		(*LogTrig(); *)
		PLC_PRG.RichiestaLogDaRemoto:=TRUE;

	2: (* REARM *)
		Sys.Warning:=FALSE;
		Sys.Alarm:=FALSE;
		Sys.AlarmStop:=FALSE;

	3: (* GET INFO1 *)
		Cmd_RLen:=6;
		TxLen:=TxLen+RAWTOHEX(ADR(Plant_SN),4,ADR(TxData[TxLen]));
		TxLen:=TxLen+RAWTOHEX(ADR(Plant_SW_VER),2,ADR(TxData[TxLen]));


(*	4: (*  Scrivo i Parametri gestione Impianto   *)

			Cmd_Buf_U16:=ADR(Cmd_Buf[8]);
			DelayAllarmeTemperaturaNonRaggiunta := Cmd_Buf_U16^; 			(* Ritardo Allarme dall'avvio Caldaia*)
			Cmd_Buf_U16:=ADR(Cmd_Buf[10]);
			DeltaInterventoAllarmeTempeaturaNonRaggiuta := Cmd_Buf_U16^;	(* Delta Soglia Temperatura per Allarme Temperatura Non Raggiunta *)
			Cmd_Buf_U16:=ADR(Cmd_Buf[12]);
			OffsetSetPointManuale := Cmd_Buf_U16^; 					(* Offest Perdite Scambiatore  *)

	5: (*  Leggi i parametri gestione Impianto  *)

			Cmd_RLen:=14;
			j:=(DelayAllarmeTemperaturaNonRaggiunta);   				(* Ritardo Allarme dall'avvio Caldaia*)
			TxLen:=TxLen+RAWTOHEX(ADR(j),2,ADR(TxData[TxLen]));
			j:=(DeltaInterventoAllarmeTempeaturaNonRaggiuta);			(* Delta Soglia Temperatura per Allarme Temperatura Non Raggiunta *)
			TxLen:=TxLen+RAWTOHEX(ADR(j),2,ADR(TxData[TxLen]));
			j:=(OffsetSetPointManuale);									(* Offest Perdite Scambiatore  *)
			TxLen:=TxLen+RAWTOHEX(ADR(j),2,ADR(TxData[TxLen]));

	6: (*  Scrivo i Parametri gestione Impianto - Antigelo   *)

			Cmd_Buf_U16:=ADR(Cmd_Buf[8]);
			SogliaMinStartAntigelo := Cmd_Buf_U16^; 			(* Soglia mininma Start Antigelo *)
			Cmd_Buf_U16:=ADR(Cmd_Buf[10]);
			SogliaMinStopAntigelo := Cmd_Buf_U16^;				(* Soglia Massima Stop Antigelo *)
			Cmd_Buf_U16:=ADR(Cmd_Buf[12]);
			BitAbilitaAntigelo :=INT_TO_BOOL( Cmd_Buf_U16^); 	(* Abilitazione Antigelo  *)

	7: (*  Leggi i parametri gestione Impianto - Antigelo *)

			Cmd_RLen:=14;
			j:=(SogliaMinStartAntigelo); 							(* Soglia mininma Start Antigelo *)
			TxLen:=TxLen+RAWTOHEX(ADR(j),2,ADR(TxData[TxLen]));
			j:=(SogliaMinStopAntigelo);								(* Soglia Massima Stop Antigelo *)
			TxLen:=TxLen+RAWTOHEX(ADR(j),2,ADR(TxData[TxLen]));
			j:=BOOL_TO_INT(BitAbilitaAntigelo);						(* Abilitazione Antigelo  *)
			TxLen:=TxLen+RAWTOHEX(ADR(j),2,ADR(TxData[TxLen]));
*)

	14: (*  Imposto data e ora del PLC  *)


			Cmd_Buf_U16:=ADR(Cmd_Buf[8]);
			SetAnno:= Cmd_Buf_U16^; 												(* Anno *)
			Cmd_Buf_U16:=ADR(Cmd_Buf[10]);
			SetMese:= Cmd_Buf_U16^;												 	(* mese *)
			Cmd_Buf_U16:=ADR(Cmd_Buf[12]);
			SetGiorno:=( Cmd_Buf_U16^);											 	(* Giorno *)
			Cmd_Buf_U16:=ADR(Cmd_Buf[14]);
			SetOra:=( Cmd_Buf_U16^); 												(* ora *)
			Cmd_Buf_U16:=ADR(Cmd_Buf[16]);
			SetMinuti:= ( Cmd_Buf_U16^);										 	(* Minuti *)
			Cmd_Buf_U16:=ADR(Cmd_Buf[18]);
			SetSecondi:= ( Cmd_Buf_U16^);										 	(* secondi *)


		SysRtcSetTime((SetDataTime(SetAnno,SetMese,SetGiorno,SetOra,SetMinuti,SetSecondi)));








ELSE
	Cmd_R:=3;
END_CASE
END_ACTION
ACTION cmd_UTA:
IF Cmd_ObjIdx<1 OR Cmd_ObjIdx>6 THEN
	Cmd_R:=2;
	RETURN;
END_IF

(* Process command *)
CASE Cmd_C OF

	1:	(* Force UTA On *)
		CASE Cmd_ObjIdx OF

			1:	UTA01.UTA_RUN_REQ := TRUE;
				UTA01.UTA_STOP_REQ 	:= FALSE;
			2:	UTA02.UTA_RUN_REQ := TRUE;
				UTA02.UTA_STOP_REQ 	:= FALSE;
			3:	UTA03.UTA_RUN_REQ := TRUE;
				UTA03.UTA_STOP_REQ 	:= FALSE;
			4:	UTA04.UTA_RUN_REQ := TRUE;
				UTA04.UTA_STOP_REQ 	:= FALSE;
			5:	UTA05.UTA_RUN_REQ := TRUE;
				UTA05.UTA_STOP_REQ 	:= FALSE;
			6:	UTA06.UTA_RUN_REQ := TRUE;
				UTA06.UTA_STOP_REQ 	:= FALSE;
			7:	UTA07.UTA_RUN_REQ := TRUE;
				UTA07.UTA_STOP_REQ 	:= FALSE;
			8:	UTA08.UTA_RUN_REQ := TRUE;
				UTA08.UTA_STOP_REQ 	:= FALSE;
			9:	UTA09.UTA_RUN_REQ := TRUE;
				UTA09.UTA_STOP_REQ 	:= FALSE;
			10:	UTA10.UTA_RUN_REQ := TRUE;
				UTA10.UTA_STOP_REQ 	:= FALSE;
			12:	UTA12.UTA_RUN_REQ := TRUE;
				UTA12.UTA_STOP_REQ 	:= FALSE;
			13:	UTA13.UTA_RUN_REQ := TRUE;
				UTA13.UTA_STOP_REQ 	:= FALSE;


		END_CASE

	2:	(* Force UTA Off *)
		CASE Cmd_ObjIdx OF

			1:	UTA01.UTA_STOP_REQ := TRUE;
				UTA01.UTA_RUN_REQ	:= FALSE;
			2:	UTA02.UTA_STOP_REQ := TRUE;
				UTA02.UTA_RUN_REQ	:= FALSE;
			3:	UTA03.UTA_STOP_REQ := TRUE;
				UTA03.UTA_RUN_REQ	:= FALSE;
			4:	UTA04.UTA_STOP_REQ := TRUE;
				UTA04.UTA_RUN_REQ	:= FALSE;
			5:	UTA05.UTA_STOP_REQ := TRUE;
				UTA05.UTA_RUN_REQ	:= FALSE;
			6:	UTA06.UTA_STOP_REQ := TRUE;
				UTA06.UTA_RUN_REQ	:= FALSE;
			7:	UTA07.UTA_STOP_REQ := TRUE;
				UTA07.UTA_RUN_REQ	:= FALSE;
			8:	UTA08.UTA_STOP_REQ := TRUE;
				UTA08.UTA_RUN_REQ	:= FALSE;
			9:	UTA09.UTA_STOP_REQ := TRUE;
				UTA09.UTA_RUN_REQ	:= FALSE;
			10:	UTA10.UTA_STOP_REQ := TRUE;
				UTA10.UTA_RUN_REQ	:= FALSE;
			12:	UTA12.UTA_STOP_REQ := TRUE;
				UTA12.UTA_RUN_REQ	:= FALSE;
			13:	UTA13.UTA_STOP_REQ := TRUE;
				UTA13.UTA_RUN_REQ	:= FALSE;

		END_CASE

	3:	(* Release force *)
		CASE Cmd_ObjIdx OF

			1:	UTA01.UTA_STOP_REQ := FALSE;
				UTA01.UTA_RUN_REQ	:= FALSE;
			2:	UTA02.UTA_STOP_REQ := FALSE;
				UTA02.UTA_RUN_REQ	:= FALSE;
			3:	UTA03.UTA_STOP_REQ := FALSE;
				UTA03.UTA_RUN_REQ	:= FALSE;
			4:	UTA04.UTA_STOP_REQ := FALSE;
				UTA04.UTA_RUN_REQ	:= FALSE;
			5:	UTA05.UTA_STOP_REQ := FALSE;
				UTA05.UTA_RUN_REQ	:= FALSE;
			6:	UTA06.UTA_STOP_REQ := FALSE;
				UTA06.UTA_RUN_REQ	:= FALSE;
			7:	UTA07.UTA_STOP_REQ := FALSE;
				UTA07.UTA_RUN_REQ	:= FALSE;
			8:	UTA08.UTA_STOP_REQ := FALSE;
				UTA08.UTA_RUN_REQ	:= FALSE;
			9:	UTA09.UTA_STOP_REQ := FALSE;
				UTA09.UTA_RUN_REQ	:= FALSE;
			10:	UTA10.UTA_STOP_REQ := FALSE;
				UTA10.UTA_RUN_REQ	:= FALSE;
			12:	UTA12.UTA_STOP_REQ := FALSE;
				UTA12.UTA_RUN_REQ	:= FALSE;
			13:	UTA13.UTA_STOP_REQ := FALSE;
				UTA13.UTA_RUN_REQ	:= FALSE;
		END_CASE

(*	4: (* SET Tempi delay On Off  *)
		CASE Cmd_ObjIdx OF
			1:	Cmd_Buf_U16:=ADR(Cmd_Buf[8]);
				UTA01.OnDelay := DWORD_TO_TIME((Cmd_Buf_U16^)*60*1000); 			(* Delay ON*)
				Cmd_Buf_U16:=ADR(Cmd_Buf[10]);
				UTA01.OffDelay := DWORD_TO_TIME((Cmd_Buf_U16^)*60*1000);			(* Delay OFF *)


		END_CASE


	5: (* GET Tempi delay On Off *)
		Cmd_RLen:=4;
			CASE Cmd_ObjIdx OF


			1:	j:=DWORD_TO_WORD(TIME_TO_DWORD((UTA01.OnDelay)/60/1000));
				TxLen:=TxLen+RAWTOHEX(ADR(j),2,ADR(TxData[TxLen]));
				j:=DWORD_TO_WORD(TIME_TO_DWORD((UTA01.OffDelay)/60/1000));
				TxLen:=TxLen+RAWTOHEX(ADR(j),2,ADR(TxData[TxLen]));


		END_CASE

*)



	8: (* SET Comandi Control Mode 0 : in manule - 1 in Automatico  *)
		CASE Cmd_ObjIdx OF
			1:	Cmd_Buf_U16:=ADR(Cmd_Buf[8]);
				cmd_ControlMode_UTA01 :=DWORD_TO_BOOL(Cmd_Buf_U16^); 	(*  0 : in manule - 1 in Automaticol *)

			2:	Cmd_Buf_U16:=ADR(Cmd_Buf[8]);
				cmd_ControlMode_UTA02 :=DWORD_TO_BOOL(Cmd_Buf_U16^); 	(*  0 : in manule - 1 in Automatico *)

			3:	Cmd_Buf_U16:=ADR(Cmd_Buf[8]);
				cmd_ControlMode_UTA03 :=DWORD_TO_BOOL(Cmd_Buf_U16^); 	(*  0 : in manule - 1 in Automatico *)

			4:	Cmd_Buf_U16:=ADR(Cmd_Buf[8]);
				cmd_ControlMode_UTA04 :=DWORD_TO_BOOL(Cmd_Buf_U16^); 	(*  0 : in manule - 1 in Automatico *)

			5:	Cmd_Buf_U16:=ADR(Cmd_Buf[8]);
				cmd_ControlMode_UTA05 :=DWORD_TO_BOOL(Cmd_Buf_U16^); 	(*  0 : in manule - 1 in Automatico *)

			6:	Cmd_Buf_U16:=ADR(Cmd_Buf[8]);
				cmd_ControlMode_UTA06 :=DWORD_TO_BOOL(Cmd_Buf_U16^); 	(*  0 : in manule - 1 in Automatico *)

			7:	Cmd_Buf_U16:=ADR(Cmd_Buf[8]);
				cmd_ControlMode_UTA07 :=DWORD_TO_BOOL(Cmd_Buf_U16^); 	(*  0 : in manule - 1 in Automatico *)

			8:	Cmd_Buf_U16:=ADR(Cmd_Buf[8]);
				cmd_ControlMode_UTA08 :=DWORD_TO_BOOL(Cmd_Buf_U16^); 	(*  0 : in manule - 1 in Automatico *)

			9:	Cmd_Buf_U16:=ADR(Cmd_Buf[8]);
				cmd_ControlMode_UTA09 :=DWORD_TO_BOOL(Cmd_Buf_U16^); 	(*  0 : in manule - 1 in Automatico *)

			10:	Cmd_Buf_U16:=ADR(Cmd_Buf[8]);
				cmd_ControlMode_UTA10 :=DWORD_TO_BOOL(Cmd_Buf_U16^); 	(*  0 : in manule - 1 in Automatico *)

	(*		11:	Cmd_Buf_U16:=ADR(Cmd_Buf[8]);
				UTA11.cmd_ControlMode_UTA :=DWORD_TO_BOOL(Cmd_Buf_U16^); 	(*  0 : in manule - 1 in Automatico *) *)

			12:	Cmd_Buf_U16:=ADR(Cmd_Buf[8]);
				cmd_ControlMode_UTA12 :=DWORD_TO_BOOL(Cmd_Buf_U16^); 	(*  0 : in manule - 1 in Automatico *)

			13:	Cmd_Buf_U16:=ADR(Cmd_Buf[8]);
				cmd_ControlMode_UTA13 :=DWORD_TO_BOOL(Cmd_Buf_U16^); 	(*  0 : in manule - 1 in Automatico *)



			END_CASE

ELSE
	Cmd_R:=3;
END_CASE
END_ACTION
ACTION Command:
(* Default response OK/NODATA *)
Cmd_R:=0;
Cmd_RLen:=0;
TxLen:=16;

(* Check object *)
CASE Cmd_Obj OF

	EO_SYS:
		Cmd_SYS();

(*	EO_GRU:
		Cmd_GRU(); *)

(*	EO_PDC:
		Cmd_PDC();

	EO_CAL:
		Cmd_CAL();
*)
	EO_CRON,EO_THER:
		Cmd_CRON();

(*	EO_VRD:
		Cmd_VRD();

	EO_CIR:
		Cmd_CIR();

	EO_CIRM:
		Cmd_CIRM();

	EO_CIRD,EO_CIRDM:
		Cmd_CIRD();

	EO_CTL:
		Cmd_CTL(); *)

	EO_CHIAERMEC:
		Cmd_CHIAERMEC();

	EO_UTACOIN:
		Cmd_UTA();

	EO_POOL:
		Cmd_POOL();

ELSE
	Cmd_R:=1;
END_CASE

(* Generate response *)
IF TxLen>0 THEN
	RAWTOHEX(ADR(Cmd_Obj)	,2,ADR(TxData[ 0]));
	RAWTOHEX(ADR(Cmd_ObjIdx),2,ADR(TxData[ 4]));
	RAWTOHEX(ADR(Cmd_R)		,2,ADR(TxData[ 8]));
	RAWTOHEX(ADR(Cmd_RLen)	,2,ADR(TxData[12]));
	TxTrig:=TRUE;
END_IF
END_ACTION

(* POU Utils Functions/TCPSERVER, ST *)
FUNCTION_BLOCK TCPSERVER
(***********************************************************************************************************	*)
(* Version: 1.6                                    			          											*)
(* Date: 11.02.2011                                   					          							    *)
(***********************************************************************************************************	*)
(* WAGO Kontakttechnik GmbH Hansastr. 27 32423 Minden(Westf.)													*)
(* Tel. +0049 571/887-0 Fax. +0049 571/887-0																	*)
(* Author: VB																									*)
(***********************************************************************************************************	*)
(*Description:	A TCP server to read and write data													       		*)
(*Historie:																										*)
(*Version 1.6: 11.02.2011: Changes according to 750-880/881											 			*)
(*Version 1.5: 27.11.2008 Bugfix allow reuse port																*)
(*Version 1.4: 13.10.2008 Bugfix transmitting large data														*)
(*Version 1.3: 15.01.2007 Changes according to FW11																*)
(*Version 1.2: 09.03.2006 Changes for socket handle 0											       			*)
(*Version 1.1: 14.02.2005 Release																				*)
(***********************************************************************************************************	*)
VAR CONSTANT
	STATE_INIT     				 : BYTE:= 0;
	STATE_OPEN     				 : BYTE:= 1;
	STATE_TX       				 : BYTE:= 20;
	STATE_RX       				 : BYTE:= 30;
	STATE_CLOSE    				 : BYTE:= 40;
	STATE_ERROR_TRAP		 	 : BYTE:= 200;
END_VAR
VAR_INPUT
	xEnable    					: BOOL;	 (* Set TRUE to enable function block *)
	wPortNumber					: WORD;  (* Port *)
	tServerTimeOut				: TIME:=t#50s;
	ptSendData					: POINTER TO ARRAY[0..MAX_SEND_TCP_SERVER] OF BYTE;
	diSendCount					: DINT;
END_VAR
VAR_OUTPUT
	xClientConnected  			: BOOL:= FALSE;
	diError 					: DINT:= 0;
END_VAR
(* Status Codes -----------------------------------------
	16#8001 => No socket descriptor available 
	16#8002 => SysSockBind fails 
	16#8003 => SysSockListen fails 
	16#8004 => switching to none blocking mode fails
	16#8005 => SysSockClose() returns FALSE 
    16#8006 => SysSockConnect() fails
    16#8007 => SysSockSend() fails
	16#8008 => error state machine 
	16#8009 => timeout while waiting for data from server 
	16#0001 => server waiting for client to establish connection
------------------------------------------------------------*)
VAR_IN_OUT
	xStartSend					: BOOL;
	aReceiveBuffer				: ARRAY [0..MAX_RECEIVE_TCP_SERVER] OF BYTE;
	diReceiveCount				: DINT;
END_VAR

VAR
	m_State    					: BYTE:= 0;
	m_ReceiveBuffer				: ARRAY [0..MAX_RECEIVE_TCP_SERVER_SOCKET] OF BYTE;
	m_ServerSocket				: DINT:= SOCKET_INVALID;
	m_Socket					: DINT:= SOCKET_INVALID;
	m_AddressInfo				: SOCKADDRESS;
	m_BytesReceived				: DINT;
	m_diReturn					: DINT;
	m_xReturn					: BOOL;
	m_SizeSockadr				: DWORD;
	m_ConnectionWatchdog		: TON;
	m_Flags						: DINT;
	m_NoneBlocking   			: DINT:= 1;
	m_Blocking   				: DINT:= 0;
	i							: INT;
	m_count						: DINT;
	diOption					: DINT := 1;
	on: DINT;
END_VAR
IF xEnable THEN
	CASE m_State OF
		STATE_INIT:
			(* Create Socket *)
			m_ServerSocket:= SysSockCreate( SOCKET_AF_INET, SOCKET_STREAM, 0);
			IF m_ServerSocket = SOCKET_INVALID THEN
				(* *)
				diError:= 16#8001;
				m_State:= STATE_ERROR_TRAP;
				RETURN;
			ELSE
				;
			END_IF
			(* Address bindings *)
			(********************)
			on:=1;
			SysSockSetOption( m_ServerSocket, SOCKET_SOL, SOCKET_SO_REUSEADDR, ADR(on), SIZEOF(on) );

			m_AddressInfo.sin_family:= SOCKET_AF_INET;
			m_AddressInfo.sin_port  := SysSockHtons( wPortNumber);
			m_AddressInfo.sin_addr  := SOCKET_INADDR_ANY;
			IF NOT SysSockBind( m_ServerSocket, ADR(m_AddressInfo), SIZEOF(m_AddressInfo)) THEN
				diError:= 16#8002;
				m_State:= STATE_ERROR_TRAP;
				RETURN;
			END_IF
			(* Wait for connections *)
			(************************)
			IF NOT SysSockListen( m_ServerSocket, 1) THEN
				diError:= 16#8003;
				m_State:= STATE_ERROR_TRAP;
			END_IF

			(* Puts SOCKET in NonBlocking mode *)
			m_diReturn:= SysSockIoctl( m_ServerSocket, SOCKET_FIONBIO, ADR(m_NoneBlocking));

			m_State:= STATE_OPEN;


		STATE_OPEN: 	(* Waiting for incomming connection *)
				m_SizeSockadr:=SIZEOF(m_AddressInfo);
				m_Socket:= SysSockAccept( m_ServerSocket, ADR(m_AddressInfo), ADR(m_SizeSockadr));
				diError:=State_open;
				IF m_Socket <> SOCKET_INVALID THEN
					xClientConnected:=TRUE;
					(*Set Push-Bit:new V1.5*)
					IF ADR(%MW0)=16#30000000  OR ADR(%MW0)=16#20000000 THEN (*841 or 881*)
						SysSockSetOption(
							diSocket:=m_Socket,
							diLevel:=6,
							diOption:=SOCKET_TCP_NODELAY,
							pOptionValue:=ADR(diOption),
							diOptionLength:=SIZEOF(diOption));
					ELSE
							;
					END_IF
					SysSockIoctl( m_Socket, SOCKET_FIONBIO, ADR(m_NoneBlocking));
					m_State:= STATE_RX;
					diError:=0;
				END_IF

		STATE_RX:
					m_BytesReceived:= SysSockRecv( m_Socket, ADR(m_ReceiveBuffer), SIZEOF(m_ReceiveBuffer), 0);
					CASE m_BytesReceived OF
					-1:(*no data available or error occured*)
						m_ConnectionWatchdog(IN:=TRUE , PT:=tServerTimeOut );
						IF m_connectionWatchdog.Q THEN
							m_State:= STATE_CLOSE;
							m_ConnectionWatchdog(IN:=FALSE);(*reset connection watchdog*)
							diError := 16#8009;
						END_IF
					0:(* socket was "gracefully closed"  *)
						m_State:= STATE_CLOSE;
						diError := 16#8003;
					ELSE
						(* Copy received data into receive buffer *)
						(********************************)
						FOR i:= 0 TO DINT_TO_INT(m_BytesReceived	)-1 DO
							aReceiveBuffer[diReceiveCount]:= m_ReceiveBuffer[i];
							diReceiveCount:=(diReceiveCount+1) MOD SIZEOF(aReceiveBuffer);
						END_FOR

						m_ConnectionWatchdog(IN:=FALSE);(*reset connection watchdog*)
					END_CASE

				(*send data*)
				IF xStartSend	 THEN
					m_State := STATE_TX;
				END_IF

	STATE_TX:	 (* send TCP-message *)
		m_diReturn := SysSockSend(diSocket := m_Socket,
								  pbyBuffer := ADR(ptSendData^[m_count]),(*geändert V1.4 bisher: [0] *)
								  diBufferSize := diSendCount-m_count,
								  diFlags :=m_Flags);
		CASE m_diReturn OF
		-1:	(* ERROR or data could not yet be send (V1.3 due to new FW11) *)
			m_ConnectionWatchdog(IN:=TRUE , PT:=tServerTimeOut );
			IF m_connectionWatchdog.Q THEN
				m_State:= STATE_CLOSE;
				m_ConnectionWatchdog(IN:=FALSE);(*reset connection watchdog*)
				diError := 16#8007;
			END_IF
		0: (* socket was "gracefully closed"  *)
			m_State := STATE_CLOSE;
			diError := 16#8003;
		ELSE (* succesful *)
			m_count:=m_count+m_diReturn;
			IF m_count>=diSendCount THEN
				diError := 16#0000;
				m_State := STATE_RX;
				m_count:=0;
				xStartSend:=FALSE;
			END_IF
			m_ConnectionWatchdog(IN:=FALSE);(*reset connection watchdog*)
		END_CASE


		STATE_CLOSE:	(* Close the server *)

